// SIMATIC S7-200 SMART project (STEP 7-Micro/WIN SMART), CPU SR30

SYMBOL_TABLE M区域
自动启停1            M0.0
手动模式1            M0.1
自动模式1            M0.2
顺序启中间1           M0.3
顺序停中间1           M0.4
自动运行状态1          M0.5
故障复位1            M0.6
自动启停2            M1.0
手动模式2            M1.1
自动模式2            M1.2
顺序启中间2           M1.3
顺序停中间2           M1.4
自动运行状态2          M1.5
故障复位2            M1.6
自动启停3            M2.0
手动模式3            M2.1
自动模式3            M2.2
顺序启中间3           M2.3
顺序停中间3           M2.4
自动运行状态3          M2.5
故障复位3            M2.6
自动启停4            M3.0     // 手动按钮启
手动模式4            M3.1
自动模式4            M3.2
顺序启中间4           M3.3
顺序停中间4           M3.4
自动运行状态4          M3.5
故障复位4            M3.6
自动启停5            M4.0
手动模式5            M4.1
自动模式5            M4.2
顺序启中间5           M4.3
顺序停中间5           M4.4
自动运行状态5          M4.5
故障复位5            M4.6
进料管破1SD          M5.0
进料管破2SD          M5.1
引风机SD            M5.2
脉冲仪1SD           M5.3
脉冲仪2SD           M5.4
脉冲仪3SD           M5.5
仓泵1出口阀1SD        M5.6
仓泵1出口阀2SD        M5.7
仓泵1呼吸阀SD         M6.0
仓泵1进料阀SD         M6.1
仓泵1进料阀上SD        M6.2
仓泵1仓顶阀SD         M6.3
仓泵1流化阀SD         M6.4
仓泵1输送阀SD         M6.5
仓泵2出口阀1SD        M6.6
仓泵2出口阀2SD        M6.7
仓泵2呼吸阀SD         M7.0
仓泵2进料阀SD         M7.1
仓泵2进料阀上SD        M7.2
仓泵2仓顶阀SD         M7.3
仓泵2流化阀SD         M7.4
仓泵2输送阀SD         M7.5
向上游要料信号1SD       M7.6
向上游要料信号2SD       M7.7
人工抽料阀SD          M9.0
人工抽料通风阀SD        M9.1
人工抽料进口阀1SD       M9.2
人工抽料进口阀2SD       M9.3
人工抽料进口阀3SD       M9.4
人工负压风机SD         M9.5
进料管破1ZD          M15.0    // 自动标志
进料管破2ZD          M15.1
引风机ZD            M15.2
仓泵1出口阀1ZD        M15.6
仓泵1出口阀2ZD        M15.7
仓泵1呼吸阀ZD         M16.0
仓泵1进料阀ZD         M16.1
仓泵1进料阀上ZD        M16.2
仓泵1仓顶阀ZD         M16.3
仓泵1流化阀ZD         M16.4
仓泵1输送阀ZD         M16.5
仓泵2出口阀1ZD        M16.6
仓泵2出口阀2ZD        M16.7
仓泵2呼吸阀ZD         M17.0
仓泵2进料阀ZD         M17.1
仓泵2进料阀上ZD        M17.2
仓泵2仓顶阀ZD         M17.3
仓泵2流化阀ZD         M17.4
仓泵2输送阀ZD         M17.5
仓泵3出口阀1ZD        M17.6
仓泵3出口阀ZD         M17.7
仓泵3呼吸阀ZD         M18.0
仓泵3进料阀ZD         M18.1
仓泵3进料阀上ZD        M18.2
仓泵3仓顶阀ZD         M18.3
仓泵3流化阀ZD         M18.4
仓泵3输送阀ZD         M18.5
仓泵2出口阀ZD         M18.6
仓泵1出口阀ZD         M18.7
仓泵4出口阀ZD         M19.0
仓泵4呼吸阀ZD         M19.1
仓泵4进料阀ZD         M19.2
仓泵4进料阀上ZD        M19.3
仓泵4仓顶阀ZD         M19.4
仓泵4流化阀ZD         M19.5
仓泵4输送阀ZD         M19.6
仓泵5出口阀ZD         M19.7
仓泵5呼吸阀ZD         M20.0
仓泵5进料阀ZD         M20.1
仓泵5进料阀上ZD        M20.2
仓泵5仓顶阀ZD         M20.3
仓泵5流化阀ZD         M20.4
仓泵5输送阀ZD         M20.5
进口阀1ZD           M21.0
出口阀1ZD           M21.1
脉冲仪1ZD           M21.2
进口阀2ZD           M21.3
出口阀2ZD           M21.4
脉冲仪2ZD           M21.5
进口阀3ZD           M21.6
出口阀3ZD           M21.7
脉冲仪3ZD           M22.0
进口阀4ZD           M22.1
出口阀4ZD           M22.2
脉冲仪4ZD           M22.3
许可按钮             M25.0
除尘器切换中           M25.7
除尘器1剔除           M26.0
除尘器2剔除           M26.1
除尘器3剔除           M26.2
除尘器4剔除           M26.3
仓泵1进料            M27.0
仓泵1出料            M27.1
仓泵1等待            M27.2
仓泵2进料            M27.3
仓泵2出料            M27.4
仓泵2等待            M27.5
仓泵3进料            M27.6
仓泵3出料            M27.7
仓泵3等待            M28.0
仓泵4进料            M28.1
仓泵4出料            M28.2
仓泵4等待            M28.3
仓泵5进料            M28.4
仓泵5出料            M28.5
仓泵5等待            M28.6
累计时间复位           M29.7
风机切换按钮           M30.0
风机切换状态           M30.1
除尘器1运行           V0.0
除尘器1停止           V0.1
除尘器1满料           V0.2
除尘器1禁止进料         V0.3
进口阀1ZJ           V0.4
出口阀1ZJ           V0.5
脉冲仪1ZJ           V0.6
仓泵禁止切换1          V0.7
除尘器2运行           V1.0
除尘器2停止           V1.1
除尘器2满料           V1.2
除尘器2禁止进料         V1.3
进口阀2ZJ           V1.4
出口阀2ZJ           V1.5
脉冲仪2ZJ           V1.6
仓泵禁止切换2          V1.7
除尘器3运行           V2.0
除尘器3停止           V2.1
除尘器3满料           V2.2
除尘器3禁止进料         V2.3
进口阀3ZJ           V2.4
出口阀3ZJ           V2.5
脉冲仪3ZJ           V2.6
仓泵禁止切换3          V2.7
除尘器4运行           V3.0
除尘器4停止           V3.1
除尘器4满料           V3.2
除尘器4禁止进料         V3.3
进口阀4ZJ           V3.4
出口阀4ZJ           V3.5
脉冲仪4ZJ           V3.6
仓泵禁止切换4          V3.7
仓泵1出口阀ZJ         V5.0
仓泵1呼吸阀ZJ         V5.1
仓泵1进料阀ZJ         V5.2
仓泵1进料阀上ZJ        V5.3
仓泵1仓顶阀ZJ         V5.4
仓泵1流化阀ZJ         V5.5
仓泵1输送阀ZJ         V5.6
仓泵1禁止输送          V5.7
仓泵2出口阀ZJ         V6.0
仓泵2呼吸阀ZJ         V6.1
仓泵2进料阀ZJ         V6.2
仓泵2进料阀上ZJ        V6.3
仓泵2仓顶阀ZJ         V6.4
仓泵2流化阀ZJ         V6.5
仓泵2输送阀ZJ         V6.6
仓泵2禁止输送          V6.7
仓泵3出口阀ZJ         V7.0
仓泵3呼吸阀ZJ         V7.1
仓泵3进料阀ZJ         V7.2
仓泵3进料阀上ZJ        V7.3
仓泵3仓顶阀ZJ         V7.4
仓泵3流化阀ZJ         V7.5
仓泵3输送阀ZJ         V7.6
仓泵3禁止输送          V7.7
仓泵4出口阀ZJ         V8.0
仓泵4呼吸阀ZJ         V8.1
仓泵4进料阀ZJ         V8.2
仓泵4进料阀上ZJ        V8.3
仓泵4仓顶阀ZJ         V8.4
仓泵4流化阀ZJ         V8.5
仓泵4输送阀ZJ         V8.6
仓泵4禁止输送          V8.7
仓泵5出口阀ZJ         V9.0
仓泵5呼吸阀ZJ         V9.1
仓泵5进料阀ZJ         V9.2
仓泵5进料阀上ZJ        V9.3
仓泵5仓顶阀ZJ         V9.4
仓泵5流化阀ZJ         V9.5
仓泵5输送阀ZJ         V9.6
仓泵5禁止输送          V9.7
急停故障M            V15.0    // 急停故障 系统1
急停_V             V15.1
                 V17.0    // 系统2
                 V18.0    // 系统3
系统3总故障M          V19.5
系统2总故障M          V19.6
系统1总故障M          V19.7
AI1_ER0          V20.0    // 系统1报警
AI1_ER1          V20.1
AI1_ER2          V20.2
AI1_ER3          V20.3
AI1_ER4          V20.4
AI1_ER5          V20.5
AI1_ER6          V20.6
AI1_ER7          V20.7
AI2_ER0          V21.0    // 系统2报警
AI2_ER1          V21.1
AI2_ER2          V21.2
AI2_ER3          V21.3
AI2_ER4          V21.4
AI2_ER5          V21.5
AI2_ER6          V21.6
AI2_ER7          V21.7
AI3_ER0          V22.0    // 系统3报警
AI3_ER1          V22.1
AI3_ER2          V22.2
AI3_ER3          V22.3
AI3_ER4          V22.4
AI3_ER5          V22.5
AI3_ER6          V22.6
AI3_ER7          V22.7
AI4_ER0          V23.0    // 备用报警
AI4_ER1          V23.1
AI4_ER2          V23.2
AI4_ER3          V23.3
AI4_ER4          V23.4
AI4_ER5          V23.5
AI4_ER6          V23.6
AI4_ER7          V23.7
AI1_ST0          V24.0    // 系统1报警
AI1_ST1          V24.1
AI1_ST2          V24.2
AI1_ST3          V24.3
AI1_ST4          V24.4
AI1_ST5          V24.5
AI1_ST6          V24.6
AI1_ST7          V24.7
AI2_ST0          V25.0    // 系统2报警
AI2_ST1          V25.1
AI2_ST2          V25.2
AI2_ST3          V25.3
AI2_ST4          V25.4
AI2_ST5          V25.5
AI2_ST6          V25.6
AI2_ST7          V25.7
AI3_ST0          V26.0    // 系统3报警
AI3_ST1          V26.1
AI3_ST2          V26.2
AI3_ST3          V26.3
AI3_ST4          V26.4
AI3_ST5          V26.5
AI3_ST6          V26.6
AI3_ST7          V26.7
AI4_ST0          V27.0    // 备用报警
AI4_ST1          V27.1
AI4_ST2          V27.2
AI4_ST3          V27.3
AI4_ST4          V27.4
AI4_ST5          V27.5
AI4_ST6          V27.6
AI4_ST7          V27.7
END_SYMBOL_TABLE

SYMBOL_TABLE 系统符号
Always_On        SM0.0    // 始终接通
First_Scan_On    SM0.1    // 仅在第一个扫描周期时接通
Clock_1s         SM0.5    // 针对 1 s 的周期时间，时钟脉冲接通 0.5 s，断开 0.5 s.
END_SYMBOL_TABLE

SYMBOL_TABLE V区域
Time1            VW200
Time2            VW202
Time3            VW204
Time4            VW206
Time5            VW208
Time6            VW210
Time7            VW212
Time8            VW214
Time9            VW216
Time10           VW218
Time11           VW220
Time12           VW222
Time13           VW224
Time14           VW226
Time15           VW228
Time16           VW230
Time17           VW232
Time18           VW234
Time19           VW236
Time20           VW238
Time21           VW240
Time22           VW242
Time23           VW244
Time24           VW246
Time25           VW248
Time26           VW250
Time27           VW252
Time28           VW254
Time29           VW256
Time30           VW258
Time31           VW260
Time32           VW262
Time33           VW264
Time34           VW266
Time35           VW268
Time36           VW270
Time37           VW272
Time38           VW274
Time39           VW276
Time40           VW278
Time41           VW280
Time42           VW282
Time43           VW284
Time44           VW286
Time45           VW288
Time46           VW290
Time47           VW292
Time48           VW294
Time49           VW296
Time50           VW298
Time51           VW300
Time52           VW302
Time53           VW304
Time54           VW306
Time55           VW308
Time56           VW310
Time57           VW312
Time58           VW314
Time59           VW316
Time60           VW318
Time61           VW320
Time62           VW322
Time63           VW324
Time64           VW326
Time65           VW328
Time66           VW330
Time67           VW332
Time68           VW334
Time69           VW336
Time70           VW338
Time71           VW340
Time72           VW342
Time73           VW344
Time74           VW346
Time75           VW348
Time76           VW350
Time77           VW352
Time78           VW354
Time79           VW356
Time80           VW358
Time81           VW360
Time82           VW362
Time83           VW364
Time84           VW366
Time85           VW368
Time86           VW370
Time87           VW372
Time88           VW374
Time89           VW376
Time90           VW378
Time91           VW380
Time92           VW382
Time93           VW384
Time94           VW386
Time95           VW388
Time96           VW390
Time97           VW392
Time98           VW394
Time99           VW396
Time100          VW398
Time101          VW400
Time102          VW402
Time103          VW404
Time104          VW406
Time105          VW408
Time106          VW410
Time107          VW412
Time108          VW414
Time109          VW416
Time110          VW418
Time111          VW420
Time112          VW422
Time113          VW424
Time114          VW426
Time115          VW428
Time116          VW430
Time117          VW432
Time118          VW434
Time119          VW436
Time120          VW438
Time121          VW440
Time122          VW442
Time123          VW444
Time124          VW446
Time125          VW448
Time126          VW450
Time127          VW452
Time128          VW454
Time129          VW456
Time130          VW458
Time131          VW460
Time132          VW462
Time133          VW464
Time134          VW466
Time135          VW468
Time136          VW470
Time137          VW472
Time138          VW474
Time139          VW476
Time140          VW478
Time141          VW480
Time142          VW482
Time143          VW484
Time144          VW486
Time145          VW488
Time146          VW490
Time147          VW492
Time148          VW494
Time149          VW496
Time150          VW498
AI_Sst_L0        VD500    // 模拟量下限0
AI_Sst_L1        VD504    // 模拟量下限1
AI_Sst_L2        VD508    // 模拟量下限2
AI_Sst_L3        VD512    // 模拟量下限3
AI_Sst_L4        VD516    // 模拟量下限4
AI_Sst_L5        VD520    // 模拟量下限5
AI_Sst_L6        VD524    // 模拟量下限6
AI_Sst_L7        VD528    // 模拟量下限7
AI_Sst_L8        VD532    // 模拟量下限8
AI_Sst_L9        VD536    // 模拟量下限9
AI_Sst_L10       VD540    // 模拟量下限10
AI_Sst_L11       VD544    // 模拟量下限11
AI_Sst_L12       VD548    // 模拟量下限12
AI_Sst_L13       VD552    // 模拟量下限13
AI_Sst_L14       VD556    // 模拟量下限14
AI_Sst_L15       VD560    // 模拟量下限15
AI_Sst_L16       VD564    // 模拟量下限16
AI_Sst_L17       VD568    // 模拟量下限17
AI_Sst_L18       VD572    // 模拟量下限18
AI_Sst_L19       VD576    // 模拟量下限19
AI_Sst_L20       VD580    // 模拟量下限20
AI_Sst_L21       VD584    // 模拟量下限21
AI_Sst_L22       VD588    // 模拟量下限22
AI_Sst_L23       VD592    // 模拟量下限23
AI_Sst_L24       VD596    // 模拟量下限24
AI_Sst_H0        VD600    // 模拟量上限0
AI_Sst_H1        VD604    // 模拟量上限1
AI_Sst_H2        VD608    // 模拟量上限2
AI_Sst_H3        VD612    // 模拟量上限3
AI_Sst_H4        VD616    // 模拟量上限4
AI_Sst_H5        VD620    // 模拟量上限5
AI_Sst_H6        VD624    // 模拟量上限6
AI_Sst_H7        VD628    // 模拟量上限7
AI_Sst_H8        VD632    // 模拟量上限8
AI_Sst_H9        VD636    // 模拟量上限9
AI_Sst_H10       VD640    // 模拟量上限10
AI_Sst_H11       VD644    // 模拟量上限11
AI_Sst_H12       VD648    // 模拟量上限12
AI_Sst_H13       VD652    // 模拟量上限13
AI_Sst_H14       VD656    // 模拟量上限14
AI_Sst_H15       VD660    // 模拟量上限15
AI_Sst_H16       VD664    // 模拟量上限16
AI_Sst_H17       VD668    // 模拟量上限17
AI_Sst_H18       VD672    // 模拟量上限18
AI_Sst_H19       VD676    // 模拟量上限19
AI_Sst_H20       VD680    // 模拟量上限20
AI_Sst_H21       VD684    // 模拟量上限21
AI_Sst_H22       VD688    // 模拟量上限22
AI_Sst_H23       VD692    // 模拟量上限23
AI_Sst_H24       VD696    // 模拟量上限24
AI_BJ_0          VD700    // 模拟量报警0
AI_BJ_1          VD704    // 模拟量报警1
AI_BJ_2          VD708    // 模拟量报警2
AI_BJ_3          VD712    // 模拟量报警3
AI_BJ_4          VD716    // 模拟量报警4
AI_BJ_5          VD720    // 模拟量报警5
AI_BJ_6          VD724    // 模拟量报警6
AI_BJ_7          VD728    // 模拟量报警7
AI_BJ_8          VD732    // 模拟量报警8
AI_BJ_9          VD736    // 模拟量报警9
AI_BJ_10         VD740    // 模拟量报警10
AI_BJ_11         VD744    // 模拟量报警11
AI_BJ_12         VD748    // 模拟量报警12
AI_BJ_13         VD752    // 模拟量报警13
AI_BJ_14         VD756    // 模拟量报警14
AI_BJ_15         VD760    // 模拟量报警15
AI_BJ_16         VD764    // 模拟量报警16
AI_BJ_17         VD768    // 模拟量报警17
AI_BJ_18         VD772    // 模拟量报警18
AI_BJ_19         VD776    // 模拟量报警19
AI_BJ_20         VD780    // 模拟量报警20
AI_BJ_21         VD784    // 模拟量报警21
AI_BJ_22         VD788    // 模拟量报警22
AI_BJ_23         VD792    // 模拟量报警23
AI_BJ_24         VD796    // 模拟量报警24
AI_TJ_0          VD800    // 模拟量停机0
AI_TJ_1          VD804    // 模拟量停机1
AI_TJ_2          VD808    // 模拟量停机2
AI_TJ_3          VD812    // 模拟量停机3
AI_TJ_4          VD816    // 模拟量停机4
AI_TJ_5          VD820    // 模拟量停机5
AI_TJ_6          VD824    // 模拟量停机6
AI_TJ_7          VD828    // 模拟量停机7
AI_TJ_8          VD832    // 模拟量停机8
AI_TJ_9          VD836    // 模拟量停机9
AI_TJ_10         VD840    // 模拟量停机10
AI_TJ_11         VD844    // 模拟量停机11
AI_TJ_12         VD848    // 模拟量停机12
AI_TJ_13         VD852    // 模拟量停机13
AI_TJ_14         VD856    // 模拟量停机14
AI_TJ_15         VD860    // 模拟量停机15
AI_TJ_16         VD864    // 模拟量停机16
AI_TJ_17         VD868    // 模拟量停机17
AI_TJ_18         VD872    // 模拟量停机18
AI_TJ_19         VD876    // 模拟量停机19
AI_TJ_20         VD880    // 模拟量停机20
AI_TJ_21         VD884    // 模拟量停机21
AI_TJ_22         VD888    // 模拟量停机22
AI_TJ_23         VD892    // 模拟量停机23
AI_TJ_24         VD896    // 模拟量停机24
AI_OUT_0         VD900    // 模拟量输出0
AI_OUT_1         VD904    // 模拟量输出1
AI_OUT_2         VD908    // 模拟量输出2
AI_OUT_3         VD912    // 模拟量输出3
AI_OUT_4         VD916    // 模拟量输出4
AI_OUT_5         VD920    // 模拟量输出5
AI_OUT_6         VD924    // 模拟量输出6
AI_OUT_7         VD928    // 模拟量输出7
AI_OUT_8         VD932    // 模拟量输出8
AI_OUT_9         VD936    // 模拟量输出9
AI_OUT_10        VD940    // 模拟量输出10
AI_OUT_11        VD944    // 模拟量输出11
AI_OUT_12        VD948    // 模拟量输出12
AI_OUT_13        VD952    // 模拟量输出13
AI_OUT_14        VD956    // 模拟量输出14
AI_OUT_15        VD960    // 模拟量输出15
AI_OUT_16        VD964    // 模拟量输出16
AI_OUT_17        VD968    // 模拟量输出17
AI_OUT_18        VD972    // 模拟量输出18
AI_OUT_19        VD976    // 模拟量输出19
AI_OUT_20        VD980    // 模拟量输出20
AI_OUT_21        VD984    // 模拟量输出21
AI_OUT_22        VD988    // 模拟量输出22
AI_OUT_23        VD992    // 模拟量输出23
AI_OUT_24        VD996    // 模拟量输出24
Set_INT_0        VW1000   // 一般整数设置
Set_INT_1        VW1002
Set_INT_2        VW1004
Set_INT_3        VW1006
Set_INT_4        VW1008
Set_INT_5        VW1010
Set_INT_6        VW1012
Set_INT_7        VW1014
Set_INT_8        VW1016
Set_INT_9        VW1018
Set_INT_10       VW1020
Set_INT_11       VW1022
Set_INT_12       VW1024
Set_INT_13       VW1026
Set_INT_14       VW1028
Out_INT_0        VW1030   // 一般整数反馈
Out_INT_1        VW1032
Out_INT_2        VW1034
Out_INT_3        VW1036
Out_INT_4        VW1038
Out_INT_5        VW1040
Out_INT_6        VW1042
Out_INT_7        VW1044
Out_INT_8        VW1046
Out_INT_9        VW1048
Out_INT_10       VW1050   // 一般整数反馈
Out_INT_11       VW1052
Out_INT_12       VW1054
Out_INT_13       VW1056
Out_INT_14       VW1058
Time_S0          VW1070   // 系统累计运行时间
Time_M0          VW1072
Time_H0          VW1074
Time_D0          VW1076
Time_S1          VW1078
Time_M1          VW1080
Time_H1          VW1082
Time_D1          VW1084
Time_S2          VW1086
Time_M2          VW1088
Time_H2          VW1090
Time_D2          VW1092
Set_R0           VD1400   // 浮点型设定
Set_R1           VD1404
Set_R2           VD1408
Set_R3           VD1412
Set_R4           VD1416
Set_R5           VD1420
Set_R6           VD1424
Set_R7           VD1428
Set_R8           VD1432
Set_R9           VD1436
Set_R10          VD1440
Set_R11          VD1444
Set_R12          VD1448
Set_R13          VD1452
Set_R14          VD1456
Set_R15          VD1460
Set_R16          VD1464
Set_R17          VD1468
Set_R18          VD1472
Set_R19          VD1476
Set_R20          VD1480
Set_R21          VD1484
Set_R22          VD1488
Set_R23          VD1492
Set_R24          VD1496
Out_R0           VD1500   // 浮点型反馈
Out_R1           VD1504
Out_R2           VD1508
Out_R3           VD1512
Out_R4           VD1516
Out_R5           VD1520
Out_R6           VD1524
Out_R7           VD1528
Out_R8           VD1532
Out_R9           VD1536
Out_R10          VD1540
Out_R11          VD1544
Out_R12          VD1548
Out_R13          VD1552
Out_R14          VD1556
Out_R15          VD1560
Out_R16          VD1564
Out_R17          VD1568
Out_R18          VD1572
Out_R19          VD1576
Out_R20          VD1580
Out_R21          VD1584
Out_R22          VD1588
Out_R23          VD1592
Out_R24          VD1596
仓泵1压力低于          VD1600
仓泵2压力低于          VD1604
仓泵3压力低于          VD1608
仓泵4压力低于          VD1612
仓泵5压力低于          VD1616
除尘器1切换值          VD1620
除尘器2切换值          VD1624
除尘器3切换值          VD1628
除尘器4切换值          VD1632
除尘器5切换值          VD1636
称重1切换值           VD1640
称重2切换值           VD1644
称重3切换值           VD1648
称重4切换值           VD1652
称重5切换值           VD1656
除尘器1设定时间         VW1660
除尘器2设定时间         VW1662
除尘器3设定时间         VW1664
除尘器4设定时间         VW1666
除尘器5设定时间         VW1668
除尘器1计时           VW1670
除尘器2计时           VW1672
除尘器3计时           VW1674
除尘器4计时           VW1676
除尘器5计时           VW1678
反打1设定时间          VW1680
反打2设定时间          VW1682
反打3设定时间          VW1684
反打4设定时间          VW1686
反打5设定时间          VW1688
反打1计时            VW1690
反打2计时            VW1692
反打3计时            VW1694
反打4计时            VW1696
反打5计时            VW1698
DINT0            VD1700
DINT1            VD1704
DINT2            VD1708
DINT3            VD1712
DINT4            VD1716
DINT5            VD1720
DINT6            VD1724
DINT7            VD1728
DINT8            VD1732
END_SYMBOL_TABLE

SYMBOL_TABLE TIMEOUT
延期执行             V1800.0
提前设定             V1800.1
密码确认             V1800.2
密码错误             V1800.3
强制冷却             V1800.4
到期               V1801.0
提前到期提醒           V1801.1
白天提醒             V1801.2
永久解锁             V1801.3
输入密码             VD1810   // 浮点数
年                VW1922
月                VW1924
日                VW1926
设定年              VW1930
设定月              VW1932
设定日              VW1934
延时月              VW1936
提前年              VW1940
提前月              VW1942
提前日              VW1944
END_SYMBOL_TABLE

SYMBOL_TABLE 通讯按需修改
控制字1             VW1100   // 通讯需要先给定047E 或者04FE
给定1              VW1102   // 十进制为 0~16384对应0~100%
控制字2             VW1110   // 由于地址冲突，不同的请从EXCL复制
给定2              VW1112   // 十进制为 0~16384对应0~100%
控制字3             VW1120   // 通讯需要先给定047E 或者04FE
给定3              VW1122   // 十进制为 0~16384对应0~100%
控制字4             VW1130   // 通讯需要先给定047E 或者04FE
给定4              VW1132   // 十进制为 0~16384对应0~100%
控制字5             VW1140   // 通讯需要先给定047E 或者04FE
给定5              VW1142   // 十进制为 0~16384对应0~100%
控制字6             VW1150   // 通讯需要先给定047E 或者04FE
给定6              VW1152   // 十进制为 0~16384对应0~100%
控制字7             VW1160   // 通讯需要先给定047E 或者04FE
给定7              VW1162   // 十进制为 0~16384对应0~100%
控制字8             VW1170   // 通讯需要先给定047E 或者04FE
给定8              VW1172   // 十进制为 0~16384对应0~100%
控制字9             VW1180   // 通讯需要先给定047E 或者04FE
给定9              VW1182   // 十进制为 0~16384对应0~100%
控制字10            VW1190   // 通讯需要先给定047E 或者04FE
给定10             VW1192   // 十进制为 0~16384对应0~100%
频率1              VW1200   // 小数点2位
电流1              VW1206   // 小数点2位
频率2              VW1210   // 小数点2位
电流2              VW1216   // 小数点2位
频率3              VW1220   // 小数点2位
电流3              VW1226   // 小数点2位
频率4              VW1230   // 小数点2位
电流4              VW1236   // 小数点2位
频率5              VW1240   // 小数点2位
电流5              VW1246   // 小数点2位
频率6              VW1250   // 小数点2位
电流6              VW1256   // 小数点2位
频率7              VW1260   // 小数点2位
电流7              VW1266   // 小数点2位
频率8              VW1270   // 小数点2位
电流8              VW1276   // 小数点2位
频率9              VW1280   // 小数点2位
电流9              VW1286   // 小数点2位
频率10             VW1290   // 小数点2位
电流10             VW1296   // 小数点2位
WC0              V60.0
WC1              V60.1
WC2              V60.2
WC3              V60.3
WC4              V60.4
WC5              V60.5
WC6              V60.6
WC7              V60.7
WC8              V61.0
WC9              V61.1
WC10             V61.2
WC11             V61.3
WC12             V61.4
WC13             V61.5
WC14             V61.6
WC15             V61.7
WC16             V62.0
WC17             V62.1
WC18             V62.2
WC19             V62.3
WC20             V62.4
切换信号             V62.7
END_SYMBOL_TABLE

SYMBOL_TABLE 仪表通讯
Uab_S            VD1310   // 施耐德仪表
Ubc_S            VD1314
Uac_S            VD1318
Ua_S             VD1322
Ub_S             VD1326
Uc_S             VD1330
Ia_S             VD1334
Ib_S             VD1338
Ic_S             VD1342
Pt_S             VD1346
EP_S             VD1350
Uab_Z            VD1360   // 以下为正泰
Ubc_Z            VD1364   // 以下为正泰
Uac_Z            VD1368   // 以下为正泰
Ua_Z             VD1372   // 以下为正泰
Ub_Z             VD1376   // 以下为正泰
Uc_Z             VD1380   // 以下为正泰
Ia_Z             VD1384   // 以下为正泰
Ib_Z             VD1388   // 以下为正泰
Ic_Z             VD1392   // 以下为正泰
Pt_Z             VD1396   // 以下为正泰
EP_Z             VD1354   // 以下为正泰
END_SYMBOL_TABLE

SYMBOL_TABLE SCR符号
仓泵1步序1           S0.0     // 步序1选择仓泵
仓泵1步序2           S0.1
仓泵1步序3           S0.2
仓泵1步序4           S0.3
仓泵1步序5           S0.4
仓泵1步序6           S0.5
仓泵2步序1           S1.0
仓泵2步序2           S1.1
仓泵2步序3           S1.2
仓泵2步序4           S1.3
仓泵2步序5           S1.4
仓泵2步序6           S1.5
仓泵3步序1           S2.0
仓泵3步序2           S2.1
仓泵3步序3           S2.2
仓泵3步序4           S2.3
仓泵3步序5           S2.4
仓泵3步序6           S2.5
仓泵4步序1           S3.0
仓泵4步序2           S3.1
仓泵4步序3           S3.2
仓泵4步序4           S3.3
仓泵4步序5           S3.4
仓泵4步序6           S3.5
仓泵5步序1           S4.0
仓泵5步序2           S4.1
仓泵5步序3           S4.2
仓泵5步序4           S4.3
仓泵5步序5           S4.4
仓泵5步序6           S4.5
END_SYMBOL_TABLE

ORGANIZATION_BLOCK MAIN:OB1
TITLE=
// 
BEGIN
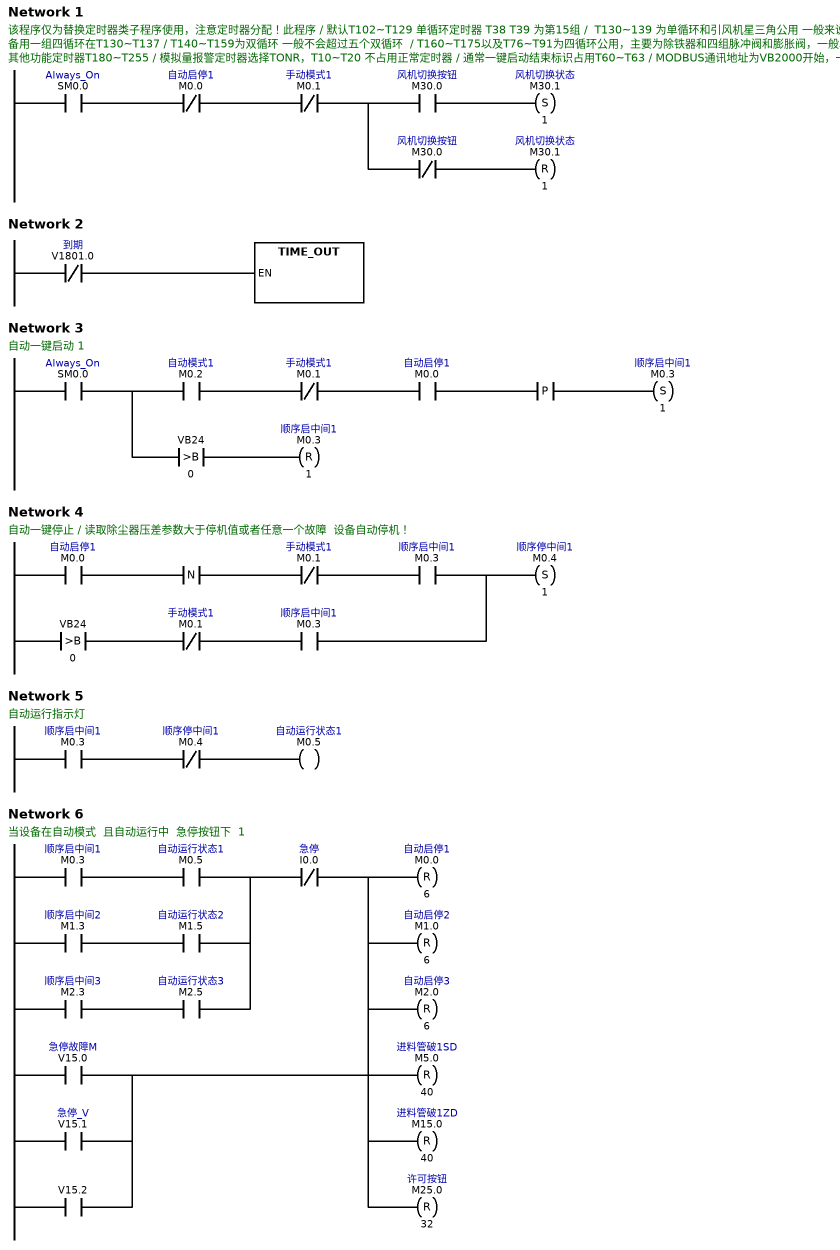
Network 1
// 该程序仅为替换定时器类子程序使用，注意定时器分配！此程序
// 默认T102~T129 单循环定时器 T38 T39 为第15组
//  T130~139 为单循环和引风机星三角公用 一般来说有星三角的程序不会用到这么多单循环阀 备用一组四循环在T130~T137
// T140~T159为双循环 一般不会超过五个双循环 
// T160~T175以及T76~T91为四循环公用，主要为除铁器和四组脉冲阀和膨胀阀，一般单独用四组
// 通常启动T40~T49 停止T50~T59 
// 其他功能定时器T180~T255
// 模拟量报警定时器选择TONR，T10~T20 不占用正常定时器
// 通常一键启动结束标识占用T60~T63
// MODBUS通讯地址为VB2000开始，一千个字节都是通讯占用区域
// 通常Time1~10为开机顺序 11~20为关机顺序 21~29为多个开关机时备用 31~80为系统仓泵或其他顺序逻辑用时间，
// Time81~120为循环时间 121~130为引风机等其他子程序时间或者循环时间备用 131~150为模拟量报警停机用
// 默认仓泵1占用T200~T214 时间31~45  仓泵2占用T215~T229 时间46~60  仓泵3占用 T230~T244 时间 61~75
// 仓泵4 占用T160~T174 时间 106~120   与四循环冲突，一般不会同时调用 与除尘器3 4 冲突
// 仓泵5占用 T175~T189 时间135~150 使用时基本会与仓泵4同时使用
// 除尘器切换主要为双除尘器 三除尘器 四除尘器 三种模式的切换子程序，只能选取一个使用
// 双除尘器切换 默认双仓泵占用 T190~T193 T46~t49  时间76~79
// 
// 
// 
LD     Always_On:SM0.0
AN     自动启停1:M0.0
AN     手动模式1:M0.1
LPS
A      风机切换按钮:M30.0
S      风机切换状态:M30.1, 1
LPP
AN     风机切换按钮:M30.0
R      风机切换状态:M30.1, 1
Network 2
LDN    到期:V1801.0
CALL   TIME_OUT:SBR5
Network 3
// 自动一键启动 1
LD     Always_On:SM0.0
LPS
A      自动模式1:M0.2
AN     手动模式1:M0.1
A      自动启停1:M0.0
EU
S      顺序启中间1:M0.3, 1
LPP
AB>    VB24, 0
R      顺序启中间1:M0.3, 1
Network 4
// 自动一键停止
// 读取除尘器压差参数大于停机值或者任意一个故障  设备自动停机！
LD     自动启停1:M0.0
ED
AN     手动模式1:M0.1
A      顺序启中间1:M0.3
LDB>   VB24, 0
AN     手动模式1:M0.1
A      顺序启中间1:M0.3
OLD
S      顺序停中间1:M0.4, 1
Network 5
// 自动运行指示灯
LD     顺序启中间1:M0.3
AN     顺序停中间1:M0.4
=      自动运行状态1:M0.5
Network 6
// 当设备在自动模式  且自动运行中  急停按钮下  1
LD     顺序启中间1:M0.3
A      自动运行状态1:M0.5
LD     顺序启中间2:M1.3
A      自动运行状态2:M1.5
OLD
LD     顺序启中间3:M2.3
A      自动运行状态3:M2.5
OLD
AN     急停:I0.0
LD     急停故障M:V15.0
O      急停_V:V15.1
O      V15.2
OLD
R      自动启停1:M0.0, 6
R      自动启停2:M1.0, 6
R      自动启停3:M2.0, 6
R      进料管破1SD:M5.0, 40
R      进料管破1ZD:M15.0, 40
R      许可按钮:M25.0, 32
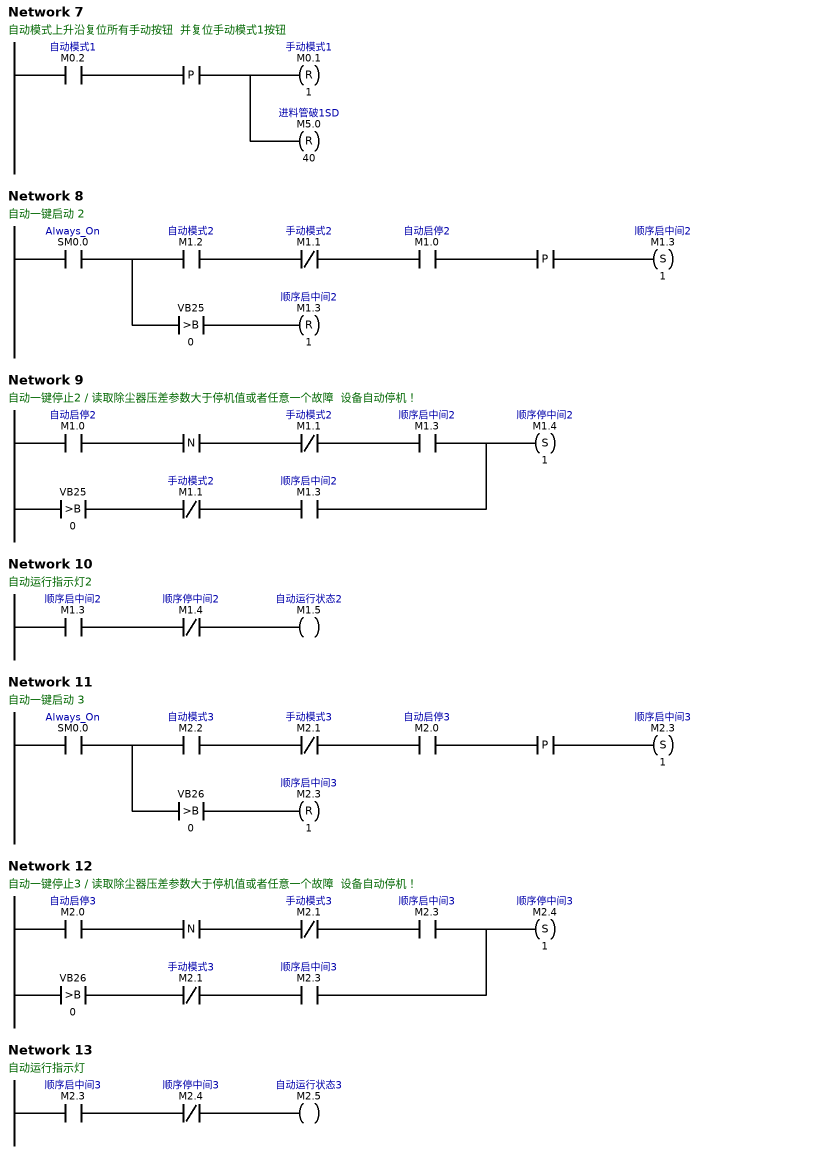
Network 7
// 自动模式上升沿复位所有手动按钮  并复位手动模式1按钮
LD     自动模式1:M0.2
EU
R      手动模式1:M0.1, 1
R      进料管破1SD:M5.0, 40
Network 8
// 自动一键启动 2
LD     Always_On:SM0.0
LPS
A      自动模式2:M1.2
AN     手动模式2:M1.1
A      自动启停2:M1.0
EU
S      顺序启中间2:M1.3, 1
LPP
AB>    VB25, 0
R      顺序启中间2:M1.3, 1
Network 9
// 自动一键停止2
// 读取除尘器压差参数大于停机值或者任意一个故障  设备自动停机！
LD     自动启停2:M1.0
ED
AN     手动模式2:M1.1
A      顺序启中间2:M1.3
LDB>   VB25, 0
AN     手动模式2:M1.1
A      顺序启中间2:M1.3
OLD
S      顺序停中间2:M1.4, 1
Network 10
// 自动运行指示灯2
LD     顺序启中间2:M1.3
AN     顺序停中间2:M1.4
=      自动运行状态2:M1.5
Network 11
// 自动一键启动 3
LD     Always_On:SM0.0
LPS
A      自动模式3:M2.2
AN     手动模式3:M2.1
A      自动启停3:M2.0
EU
S      顺序启中间3:M2.3, 1
LPP
AB>    VB26, 0
R      顺序启中间3:M2.3, 1
Network 12
// 自动一键停止3
// 读取除尘器压差参数大于停机值或者任意一个故障  设备自动停机！
LD     自动启停3:M2.0
ED
AN     手动模式3:M2.1
A      顺序启中间3:M2.3
LDB>   VB26, 0
AN     手动模式3:M2.1
A      顺序启中间3:M2.3
OLD
S      顺序停中间3:M2.4, 1
Network 13
// 自动运行指示灯
LD     顺序启中间3:M2.3
AN     顺序停中间3:M2.4
=      自动运行状态3:M2.5
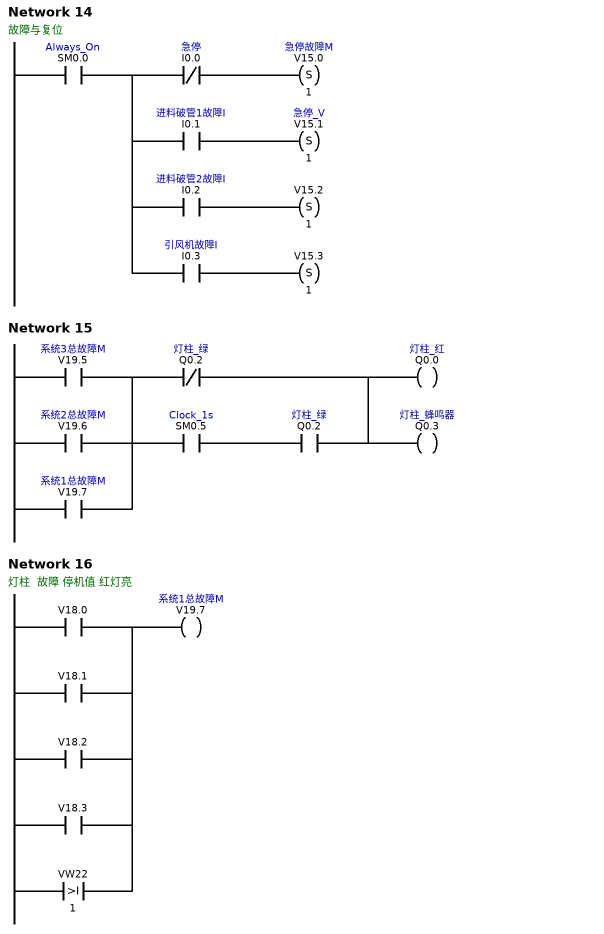
Network 14
// 故障与复位
LD     Always_On:SM0.0
LPS
AN     急停:I0.0
S      急停故障M:V15.0, 1
LRD
A      进料破管1故障I:I0.1
S      急停_V:V15.1, 1
LRD
A      进料破管2故障I:I0.2
S      V15.2, 1
LPP
A      引风机故障I:I0.3
S      V15.3, 1
Network 15
LD     系统3总故障M:V19.5
O      系统2总故障M:V19.6
O      系统1总故障M:V19.7
LDN    灯柱_绿:Q0.2
LD     Clock_1s:SM0.5
A      灯柱_绿:Q0.2
OLD
ALD
=      灯柱_红:Q0.0
=      灯柱_蜂鸣器:Q0.3
Network 16
// 灯柱  故障 停机值 红灯亮
LD     V18.0
O      V18.1
O      V18.2
O      V18.3
OW>    VW22, 1
=      系统1总故障M:V19.7
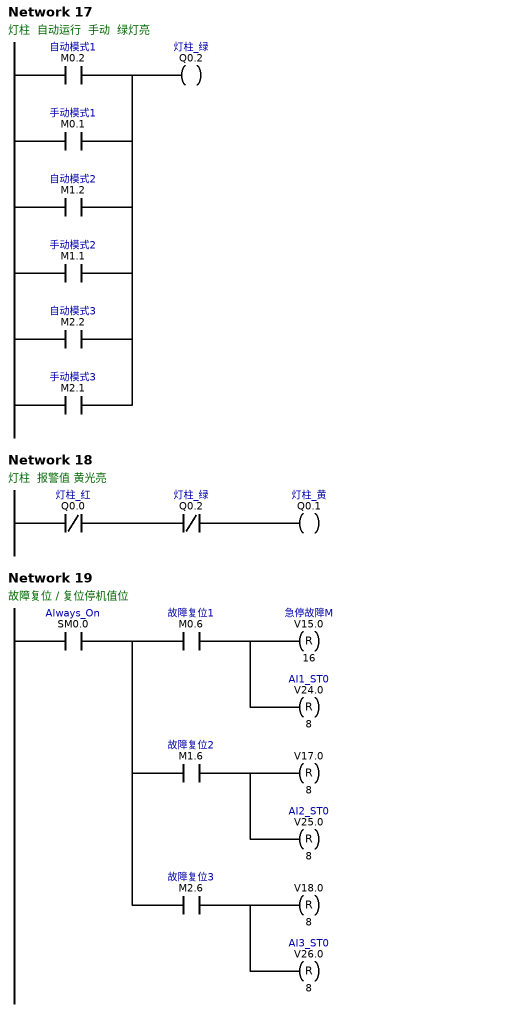
Network 17
// 灯柱  自动运行  手动  绿灯亮
LD     自动模式1:M0.2
O      手动模式1:M0.1
O      自动模式2:M1.2
O      手动模式2:M1.1
O      自动模式3:M2.2
O      手动模式3:M2.1
=      灯柱_绿:Q0.2
Network 18
// 灯柱  报警值 黄光亮
LDN    灯柱_红:Q0.0
AN     灯柱_绿:Q0.2
=      灯柱_黄:Q0.1
Network 19
// 故障复位
// 复位停机值位
LD     Always_On:SM0.0
LPS
A      故障复位1:M0.6
R      急停故障M:V15.0, 16
R      AI1_ST0:V24.0, 8
LRD
A      故障复位2:M1.6
R      V17.0, 8
R      AI2_ST0:V25.0, 8
LPP
A      故障复位3:M2.6
R      V18.0, 8
R      AI3_ST0:V26.0, 8
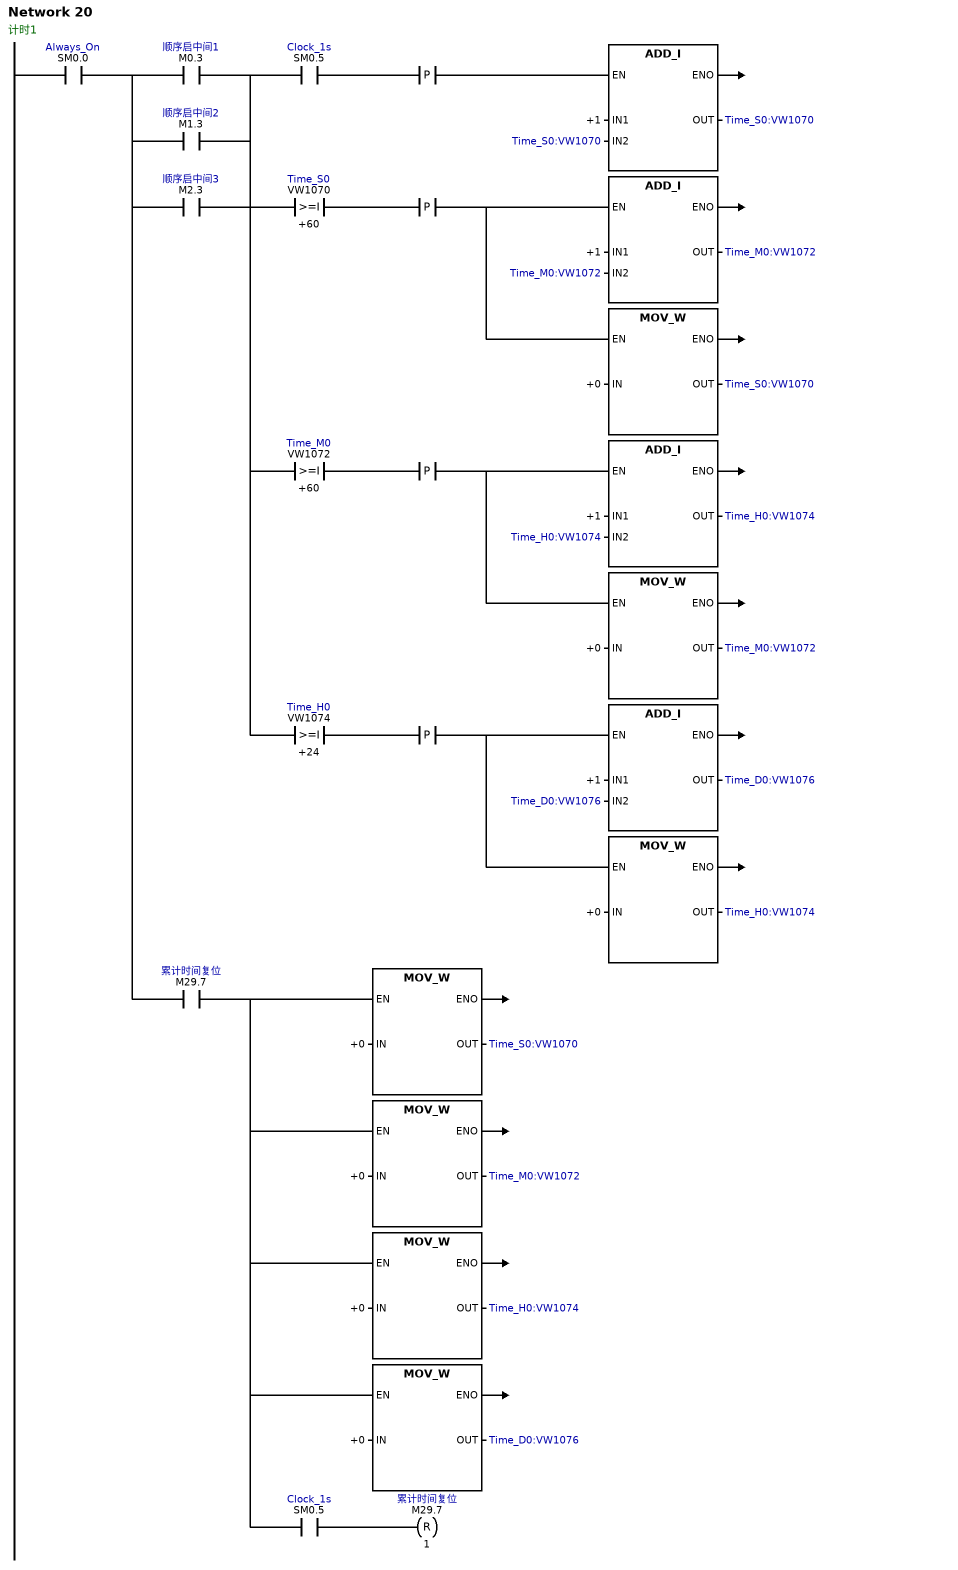
Network 20
// 计时1
LD     Always_On:SM0.0
LPS
LD     顺序启中间1:M0.3
O      顺序启中间2:M1.3
O      顺序启中间3:M2.3
ALD
LPS
A      Clock_1s:SM0.5
EU
+I     +1, Time_S0:VW1070
LRD
AW>=   Time_S0:VW1070, +60
EU
+I     +1, Time_M0:VW1072
MOVW   +0, Time_S0:VW1070
LRD
AW>=   Time_M0:VW1072, +60
EU
+I     +1, Time_H0:VW1074
MOVW   +0, Time_M0:VW1072
LPP
AW>=   Time_H0:VW1074, +24
EU
+I     +1, Time_D0:VW1076
MOVW   +0, Time_H0:VW1074
LPP
A      累计时间复位:M29.7
MOVW   +0, Time_S0:VW1070
MOVW   +0, Time_M0:VW1072
MOVW   +0, Time_H0:VW1074
MOVW   +0, Time_D0:VW1076
A      Clock_1s:SM0.5
R      累计时间复位:M29.7, 1
END_ORGANIZATION_BLOCK

// SBR0: protected block, not included

// SBR1: protected block, not included

// SBR2: protected block, not included

// SBR3: protected block, not included

// SBR4: protected block, not included

SUBROUTINE_BLOCK TIME_OUT:SBR5
TITLE=
BEGIN
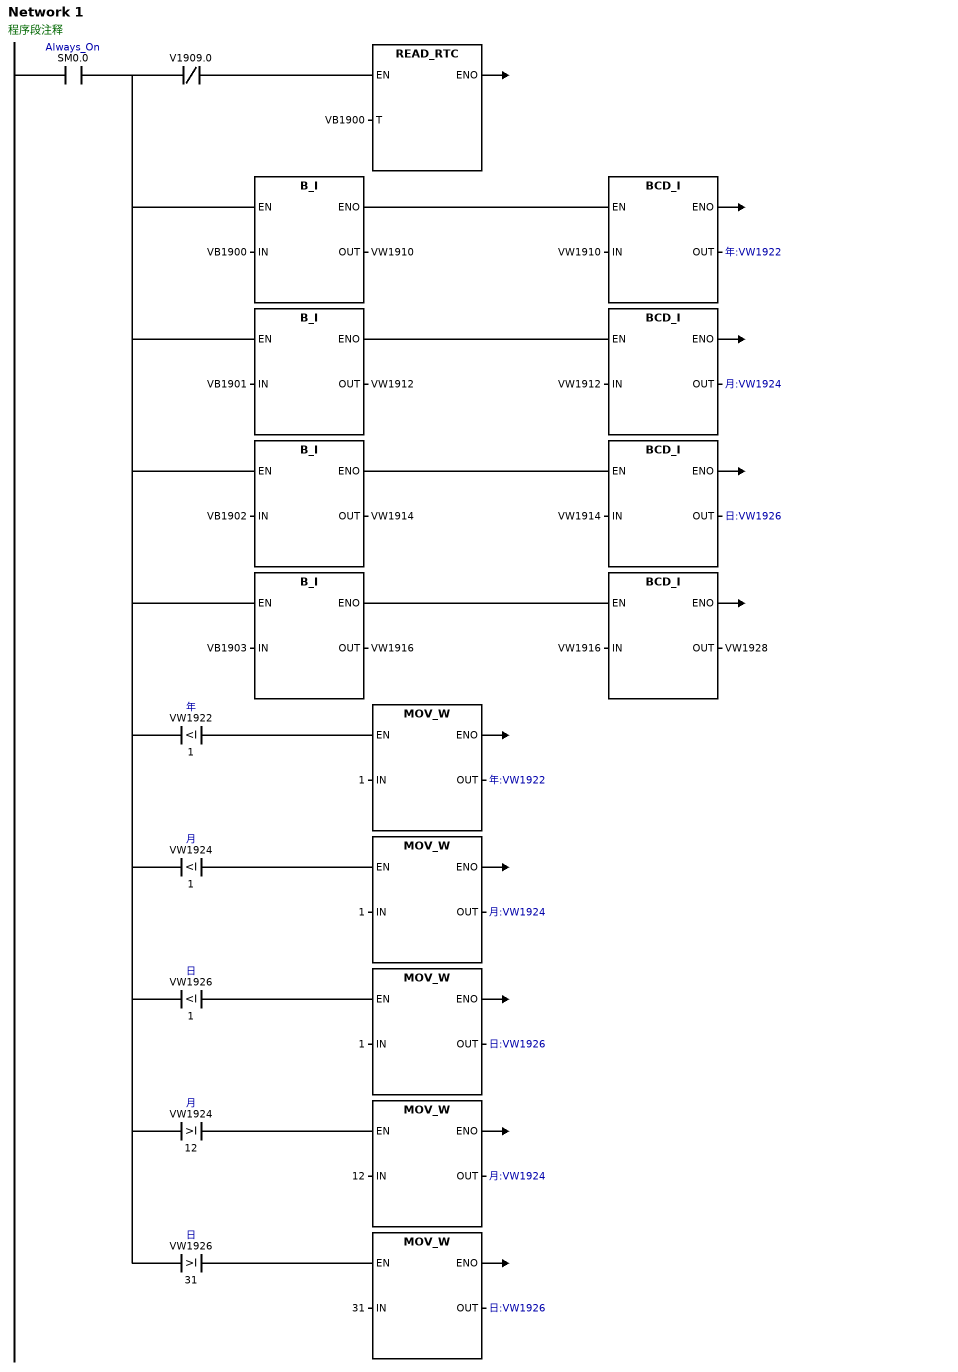
Network 1
// 程序段注释
LD     Always_On:SM0.0
LPS
AN     V1909.0
TODR   VB1900
LRD
BTI    VB1900, VW1910
AENO
MOVW   VW1910, 年:VW1922
BCDI   年:VW1922
LRD
BTI    VB1901, VW1912
AENO
MOVW   VW1912, 月:VW1924
BCDI   月:VW1924
LRD
BTI    VB1902, VW1914
AENO
MOVW   VW1914, 日:VW1926
BCDI   日:VW1926
LRD
BTI    VB1903, VW1916
AENO
MOVW   VW1916, VW1928
BCDI   VW1928
LRD
AW<    年:VW1922, 1
MOVW   1, 年:VW1922
LRD
AW<    月:VW1924, 1
MOVW   1, 月:VW1924
LRD
AW<    日:VW1926, 1
MOVW   1, 日:VW1926
LRD
AW>    月:VW1924, 12
MOVW   12, 月:VW1924
LPP
AW>    日:VW1926, 31
MOVW   31, 日:VW1926
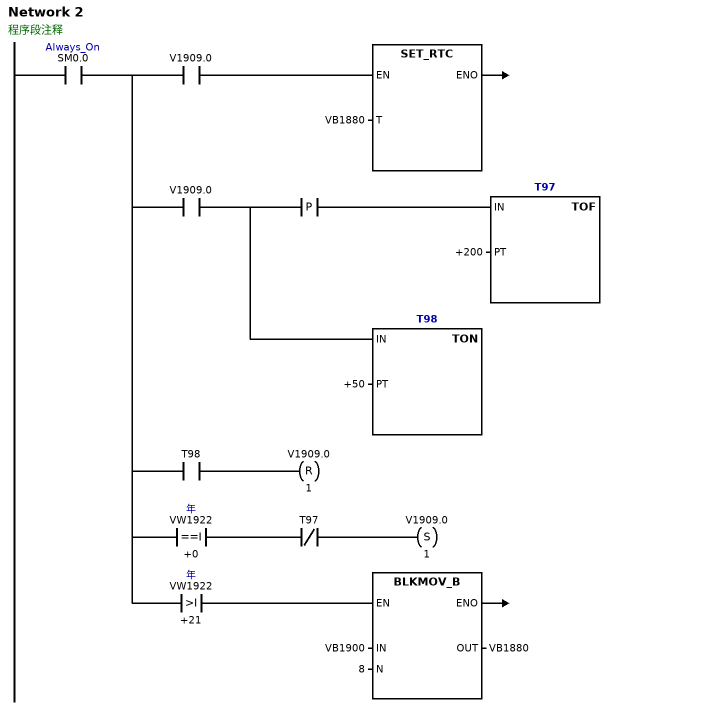
Network 2
// 程序段注释
LD     Always_On:SM0.0
LPS
A      V1909.0
TODW   VB1880
LRD
A      V1909.0
LPS
EU
TOF    T97, +200
LPP
TON    T98, +50
LPP
LPS
A      T98
R      V1909.0, 1
LRD
AW=    年:VW1922, +0
AN     T97
S      V1909.0, 1
LPP
AW>    年:VW1922, +21
BMB    VB1900, VB1880, 8
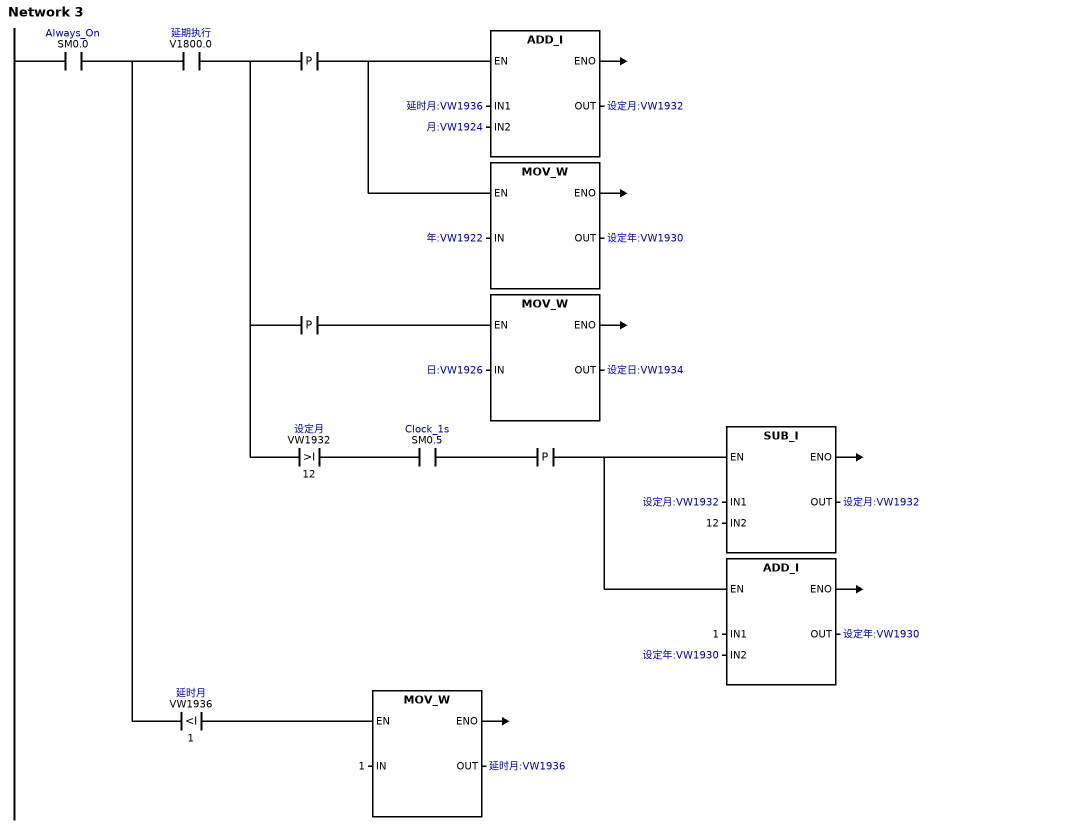
Network 3
LD     Always_On:SM0.0
LPS
A      延期执行:V1800.0
LPS
EU
MOVW   延时月:VW1936, 设定月:VW1932
+I     月:VW1924, 设定月:VW1932
MOVW   年:VW1922, 设定年:VW1930
LRD
EU
MOVW   日:VW1926, 设定日:VW1934
LPP
AW>    设定月:VW1932, 12
A      Clock_1s:SM0.5
EU
-I     12, 设定月:VW1932
+I     1, 设定年:VW1930
LPP
AW<    延时月:VW1936, 1
MOVW   1, 延时月:VW1936
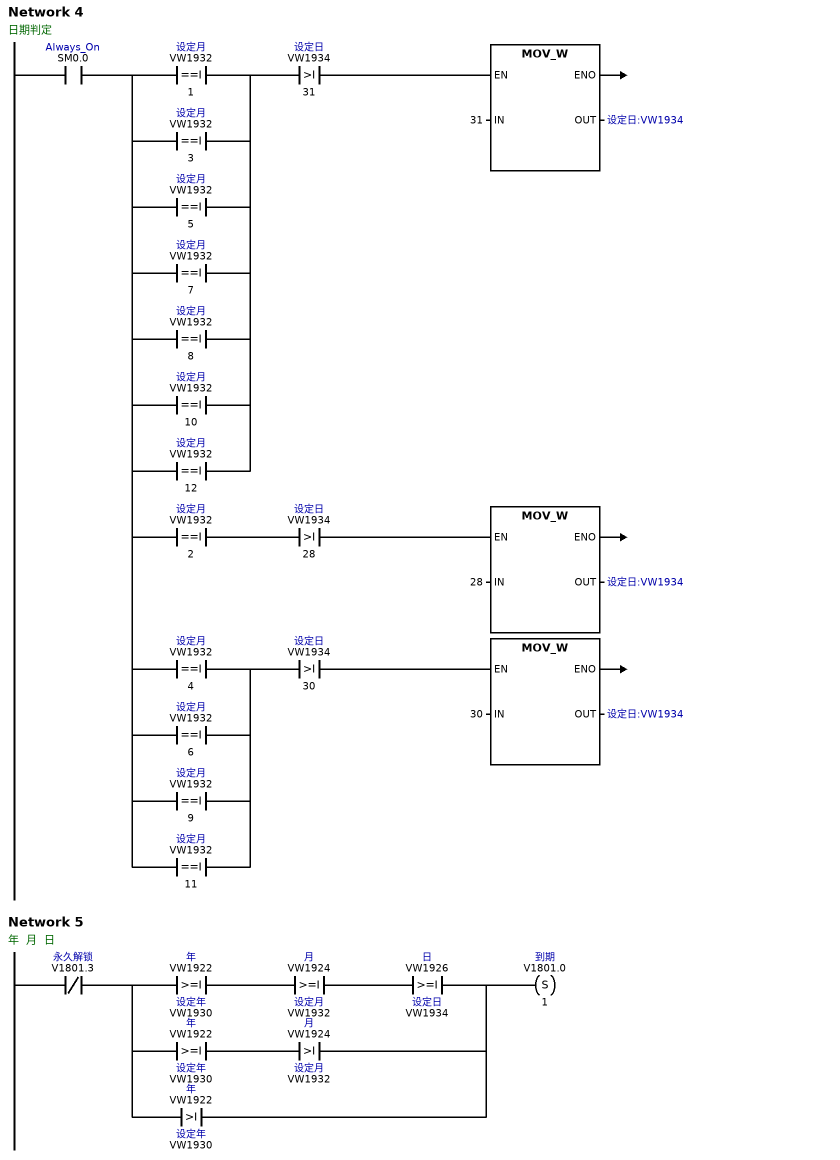
Network 4
// 日期判定
LD     Always_On:SM0.0
LPS
LDW=   设定月:VW1932, 1
OW=    设定月:VW1932, 3
OW=    设定月:VW1932, 5
OW=    设定月:VW1932, 7
OW=    设定月:VW1932, 8
OW=    设定月:VW1932, 10
OW=    设定月:VW1932, 12
ALD
AW>    设定日:VW1934, 31
MOVW   31, 设定日:VW1934
LRD
AW=    设定月:VW1932, 2
AW>    设定日:VW1934, 28
MOVW   28, 设定日:VW1934
LPP
LDW=   设定月:VW1932, 4
OW=    设定月:VW1932, 6
OW=    设定月:VW1932, 9
OW=    设定月:VW1932, 11
ALD
AW>    设定日:VW1934, 30
MOVW   30, 设定日:VW1934
Network 5
// 年  月  日 
LDN    永久解锁:V1801.3
LDW>=  年:VW1922, 设定年:VW1930
AW>=   月:VW1924, 设定月:VW1932
AW>=   日:VW1926, 设定日:VW1934
LDW>=  年:VW1922, 设定年:VW1930
AW>    月:VW1924, 设定月:VW1932
OLD
OW>    年:VW1922, 设定年:VW1930
ALD
S      到期:V1801.0, 1
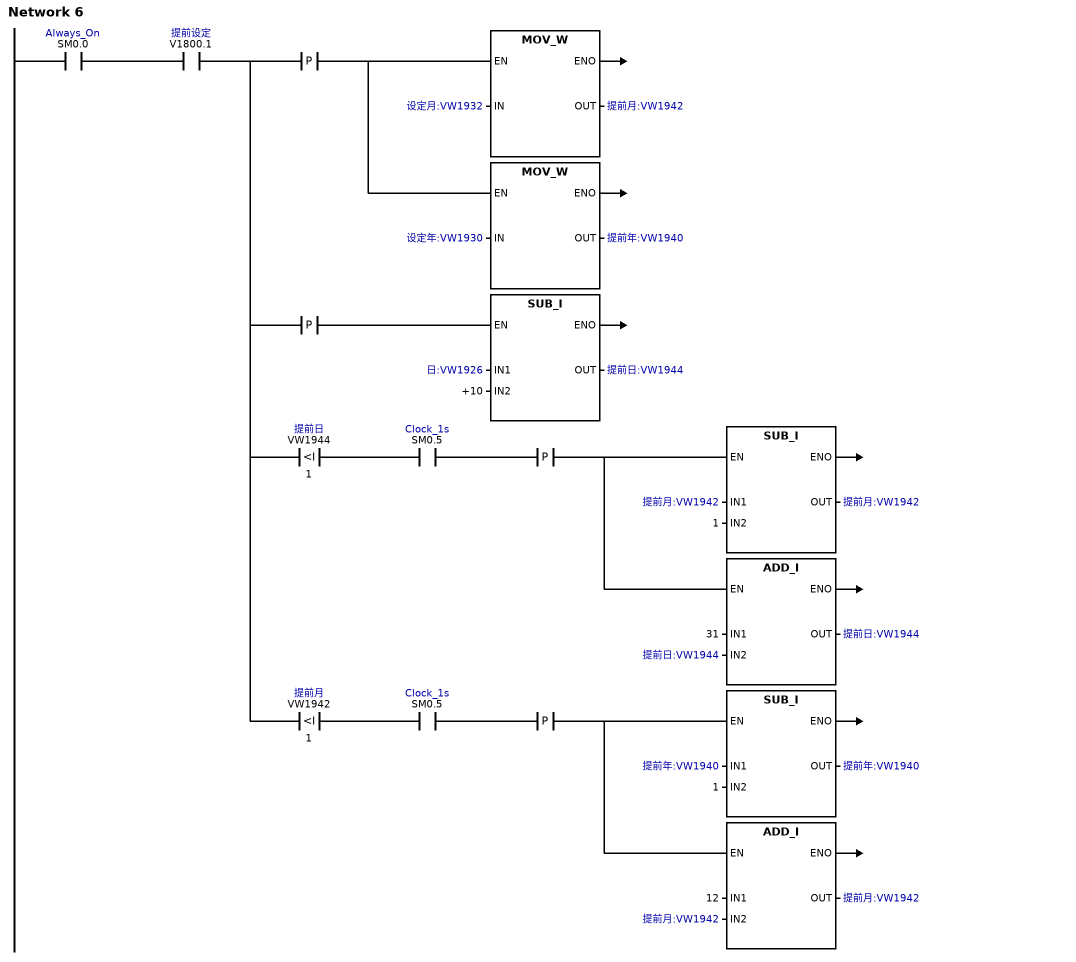
Network 6
LD     Always_On:SM0.0
A      提前设定:V1800.1
LPS
EU
MOVW   设定月:VW1932, 提前月:VW1942
MOVW   设定年:VW1930, 提前年:VW1940
LRD
EU
MOVW   日:VW1926, 提前日:VW1944
-I     +10, 提前日:VW1944
LRD
AW<    提前日:VW1944, 1
A      Clock_1s:SM0.5
EU
-I     1, 提前月:VW1942
+I     31, 提前日:VW1944
LPP
AW<    提前月:VW1942, 1
A      Clock_1s:SM0.5
EU
-I     1, 提前年:VW1940
+I     12, 提前月:VW1942
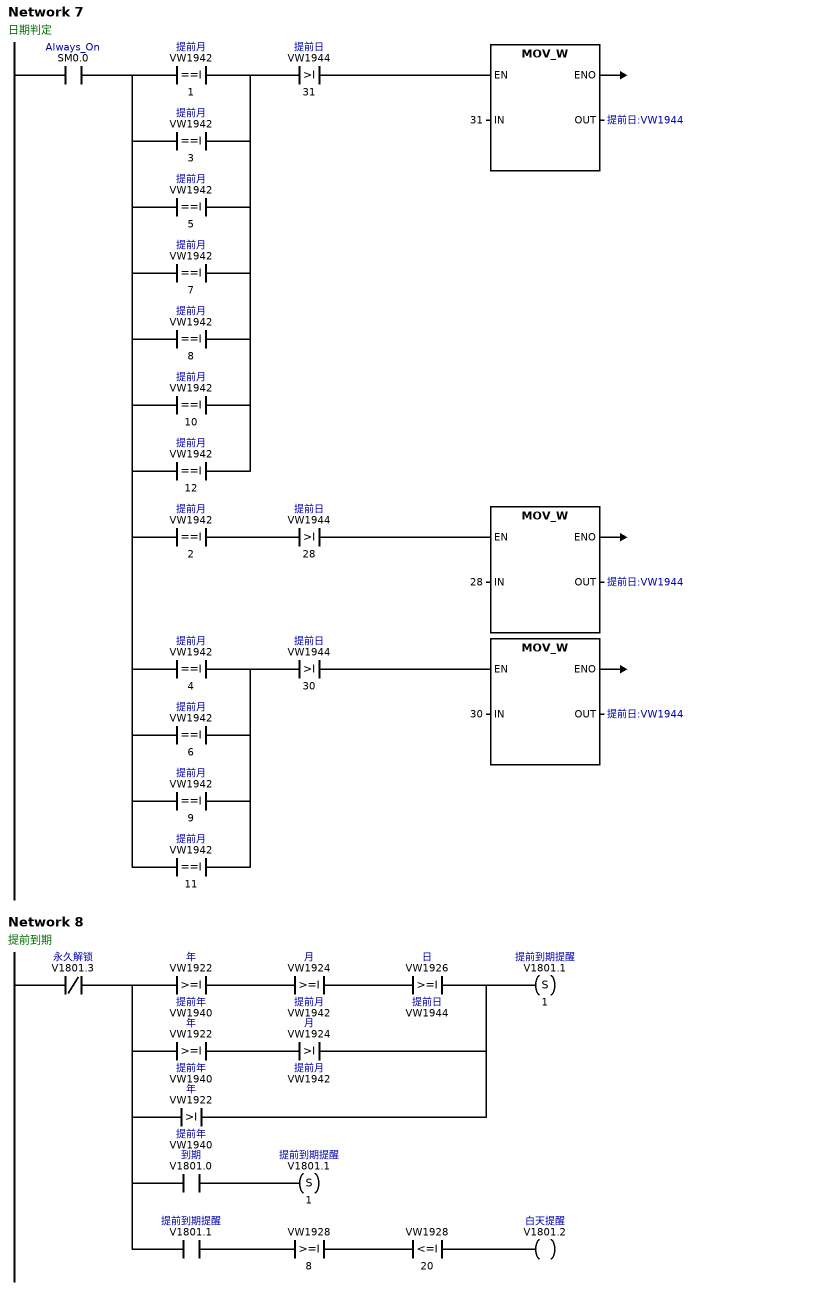
Network 7
// 日期判定
LD     Always_On:SM0.0
LPS
LDW=   提前月:VW1942, 1
OW=    提前月:VW1942, 3
OW=    提前月:VW1942, 5
OW=    提前月:VW1942, 7
OW=    提前月:VW1942, 8
OW=    提前月:VW1942, 10
OW=    提前月:VW1942, 12
ALD
AW>    提前日:VW1944, 31
MOVW   31, 提前日:VW1944
LRD
AW=    提前月:VW1942, 2
AW>    提前日:VW1944, 28
MOVW   28, 提前日:VW1944
LPP
LDW=   提前月:VW1942, 4
OW=    提前月:VW1942, 6
OW=    提前月:VW1942, 9
OW=    提前月:VW1942, 11
ALD
AW>    提前日:VW1944, 30
MOVW   30, 提前日:VW1944
Network 8
// 提前到期
LDN    永久解锁:V1801.3
LPS
LDW>=  年:VW1922, 提前年:VW1940
AW>=   月:VW1924, 提前月:VW1942
AW>=   日:VW1926, 提前日:VW1944
LDW>=  年:VW1922, 提前年:VW1940
AW>    月:VW1924, 提前月:VW1942
OLD
OW>    年:VW1922, 提前年:VW1940
ALD
S      提前到期提醒:V1801.1, 1
LPP
LPS
A      到期:V1801.0
S      提前到期提醒:V1801.1, 1
LPP
A      提前到期提醒:V1801.1
AW>=   VW1928, 8
AW<=   VW1928, 20
=      白天提醒:V1801.2
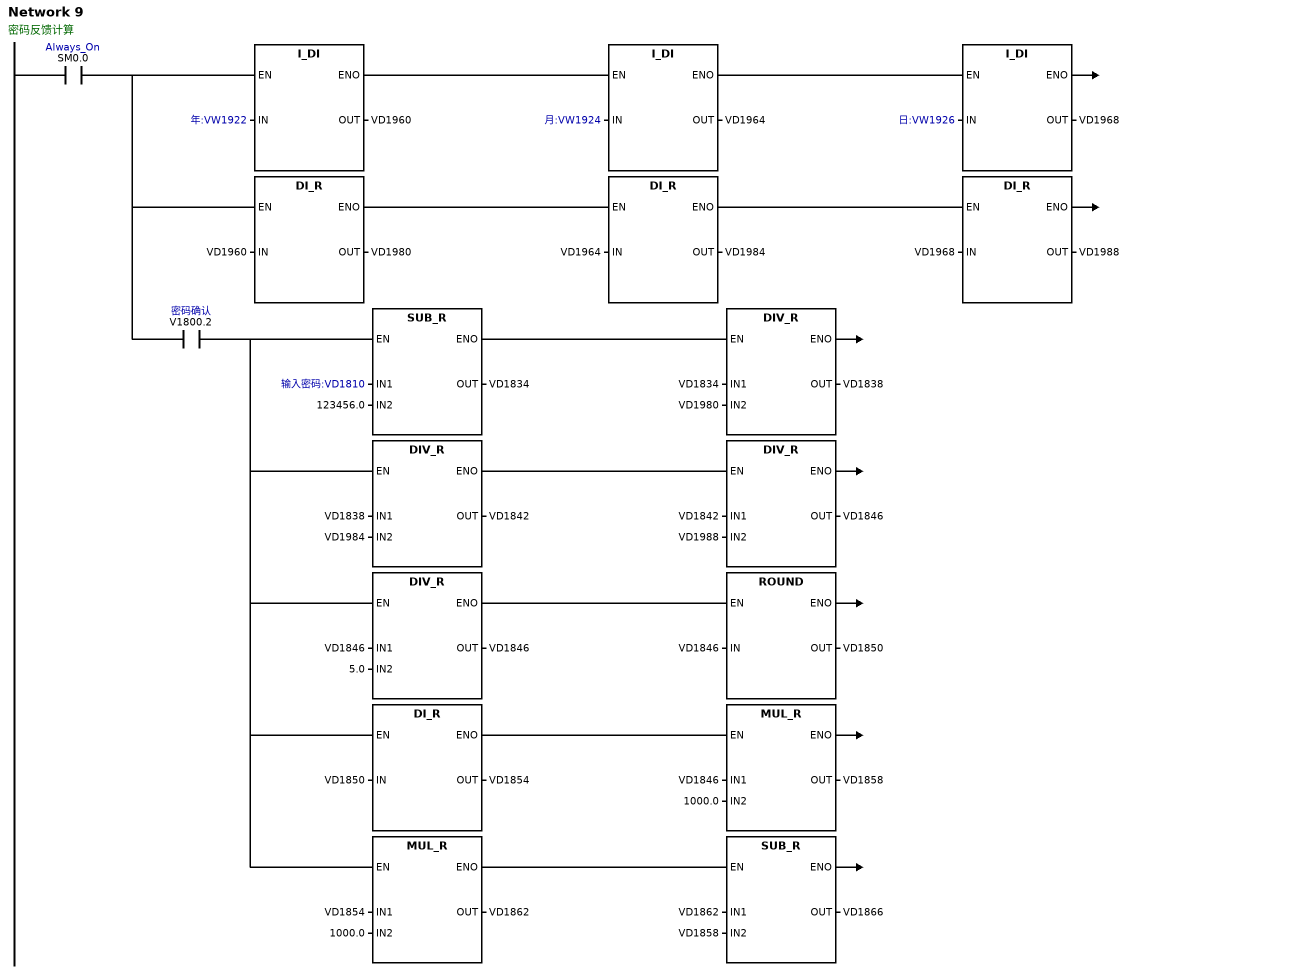
Network 9
// 密码反馈计算
LD     Always_On:SM0.0
LPS
ITD    年:VW1922, VD1960
AENO
ITD    月:VW1924, VD1964
AENO
ITD    日:VW1926, VD1968
LRD
DTR    VD1960, VD1980
AENO
DTR    VD1964, VD1984
AENO
DTR    VD1968, VD1988
LPP
A      密码确认:V1800.2
LPS
MOVR   输入密码:VD1810, VD1834
AENO
-R     123456.0, VD1834
AENO
MOVR   VD1834, VD1838
/R     VD1980, VD1838
LRD
MOVR   VD1838, VD1842
AENO
/R     VD1984, VD1842
AENO
MOVR   VD1842, VD1846
/R     VD1988, VD1846
LRD
/R     5.0, VD1846
AENO
ROUND  VD1846, VD1850
LRD
DTR    VD1850, VD1854
AENO
MOVR   VD1846, VD1858
*R     1000.0, VD1858
LPP
MOVR   VD1854, VD1862
AENO
*R     1000.0, VD1862
AENO
MOVR   VD1862, VD1866
-R     VD1858, VD1866
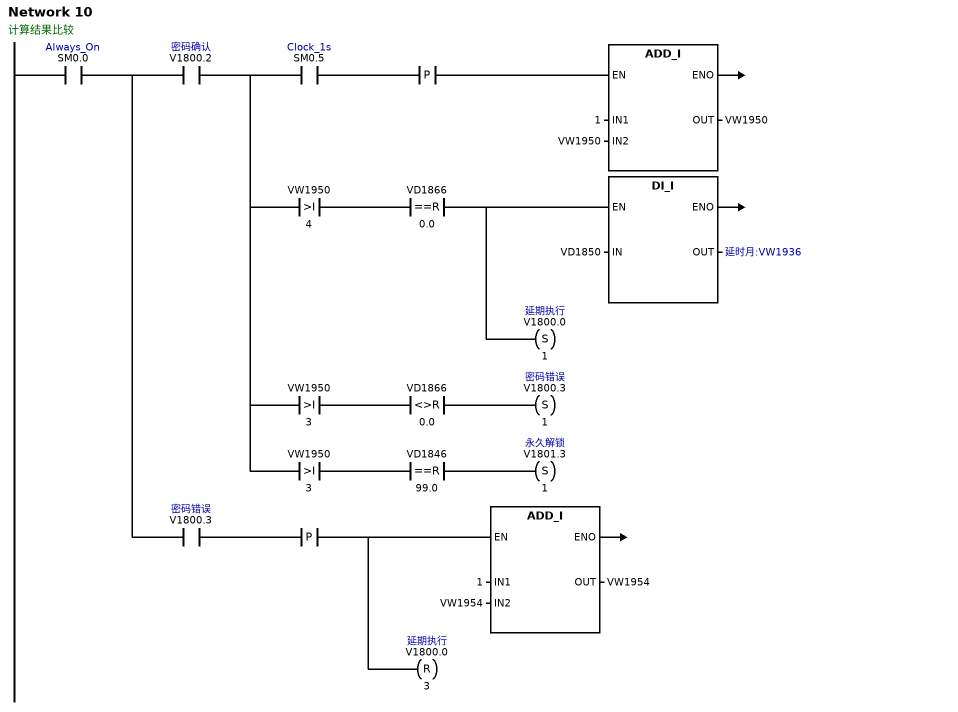
Network 10
// 计算结果比较
LD     Always_On:SM0.0
LPS
A      密码确认:V1800.2
LPS
A      Clock_1s:SM0.5
EU
+I     1, VW1950
LRD
AW>    VW1950, 4
AR=    VD1866, 0.0
DTI    VD1850, 延时月:VW1936
S      延期执行:V1800.0, 1
LPP
LPS
AW>    VW1950, 3
AR<>   VD1866, 0.0
S      密码错误:V1800.3, 1
LPP
AW>    VW1950, 3
AR=    VD1846, 99.0
S      永久解锁:V1801.3, 1
LPP
A      密码错误:V1800.3
EU
+I     1, VW1954
R      延期执行:V1800.0, 3
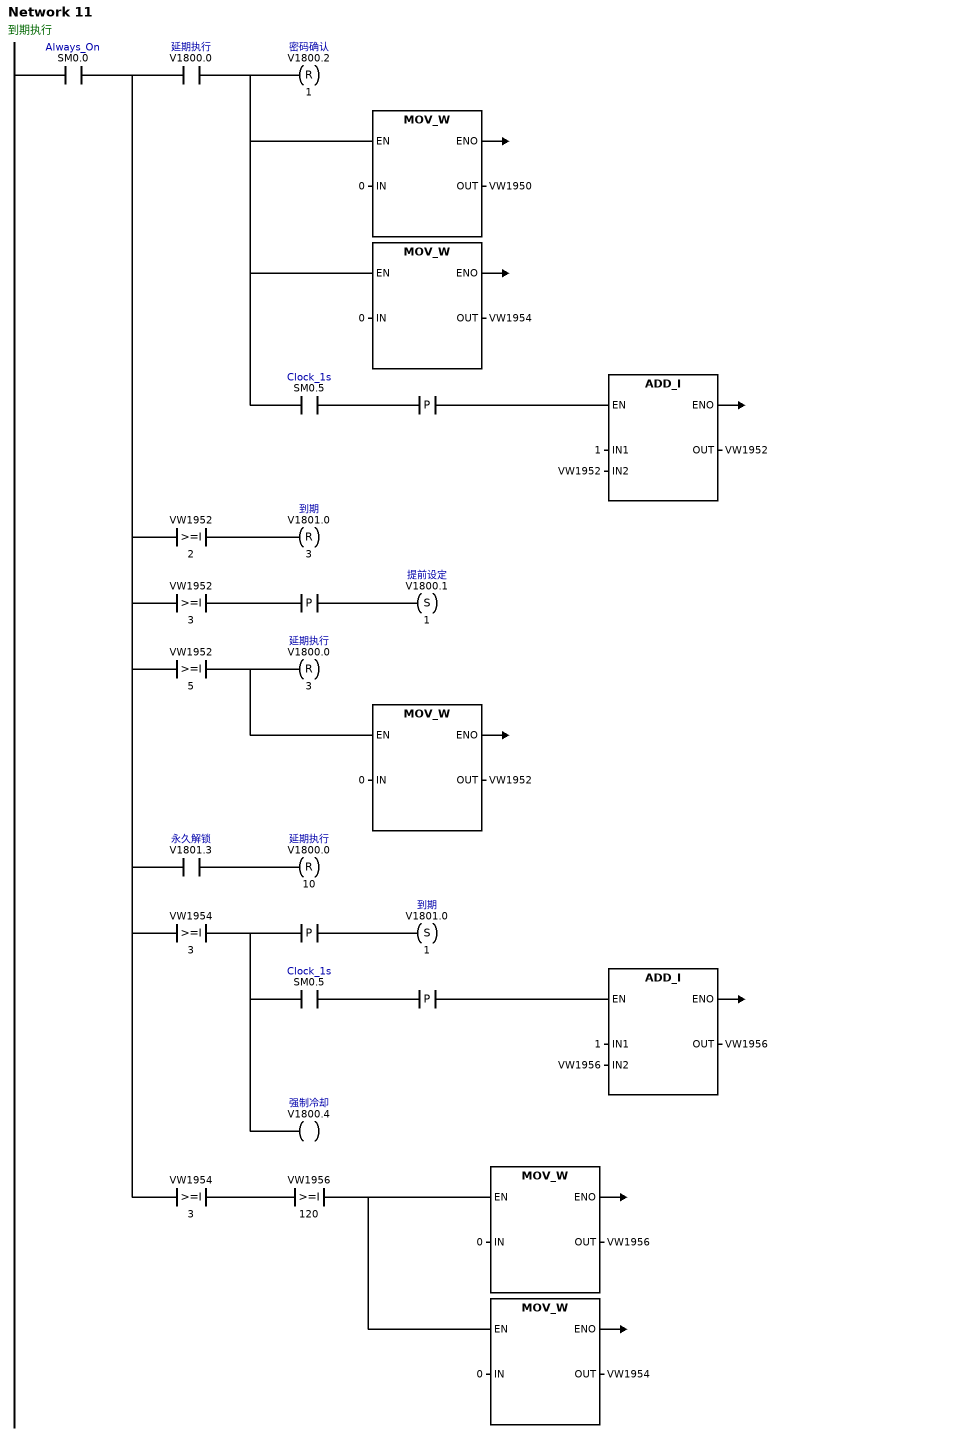
Network 11
// 到期执行
LD     Always_On:SM0.0
LPS
A      延期执行:V1800.0
R      密码确认:V1800.2, 1
MOVW   0, VW1950
MOVW   0, VW1954
A      Clock_1s:SM0.5
EU
+I     1, VW1952
LRD
LPS
AW>=   VW1952, 2
R      到期:V1801.0, 3
LPP
AW>=   VW1952, 3
EU
S      提前设定:V1800.1, 1
LRD
AW>=   VW1952, 5
R      延期执行:V1800.0, 3
MOVW   0, VW1952
LRD
A      永久解锁:V1801.3
R      延期执行:V1800.0, 10
LRD
AW>=   VW1954, 3
LPS
EU
S      到期:V1801.0, 1
LRD
A      Clock_1s:SM0.5
EU
+I     1, VW1956
LPP
=      强制冷却:V1800.4
LPP
AW>=   VW1954, 3
AW>=   VW1956, 120
MOVW   0, VW1956
MOVW   0, VW1954
END_SUBROUTINE_BLOCK

// SBR6: protected block, not included

// SBR7: protected block, not included

SUBROUTINE_BLOCK 系统按钮:SBR8
TITLE=
VAR_IN_OUT
Auto_Mode:BOOL;	// L0.0 
Hand_Mode:BOOL;	// L0.1 
System_Star:BOOL;	// L0.2 
Star_Middle:BOOL;	// L0.3 
Stop_Middle:BOOL;	// L0.4 
Auto_State:BOOL;	// L0.5 
Rest:BOOL;	// L0.6 
Standby:BOOL;	// L0.7 
Error1_Stop:BOOL;	// L1.0 
Error2_Stop:BOOL;	// L1.1 
Error3_Stop:BOOL;	// L1.2 
Error4_Stop:BOOL;	// L1.3 
System_Error:BOOL;	// L1.4 
E_Stop:BOOL;	// L1.5 
Stop_over:BOOL;	// L1.6 
END_VAR
BEGIN
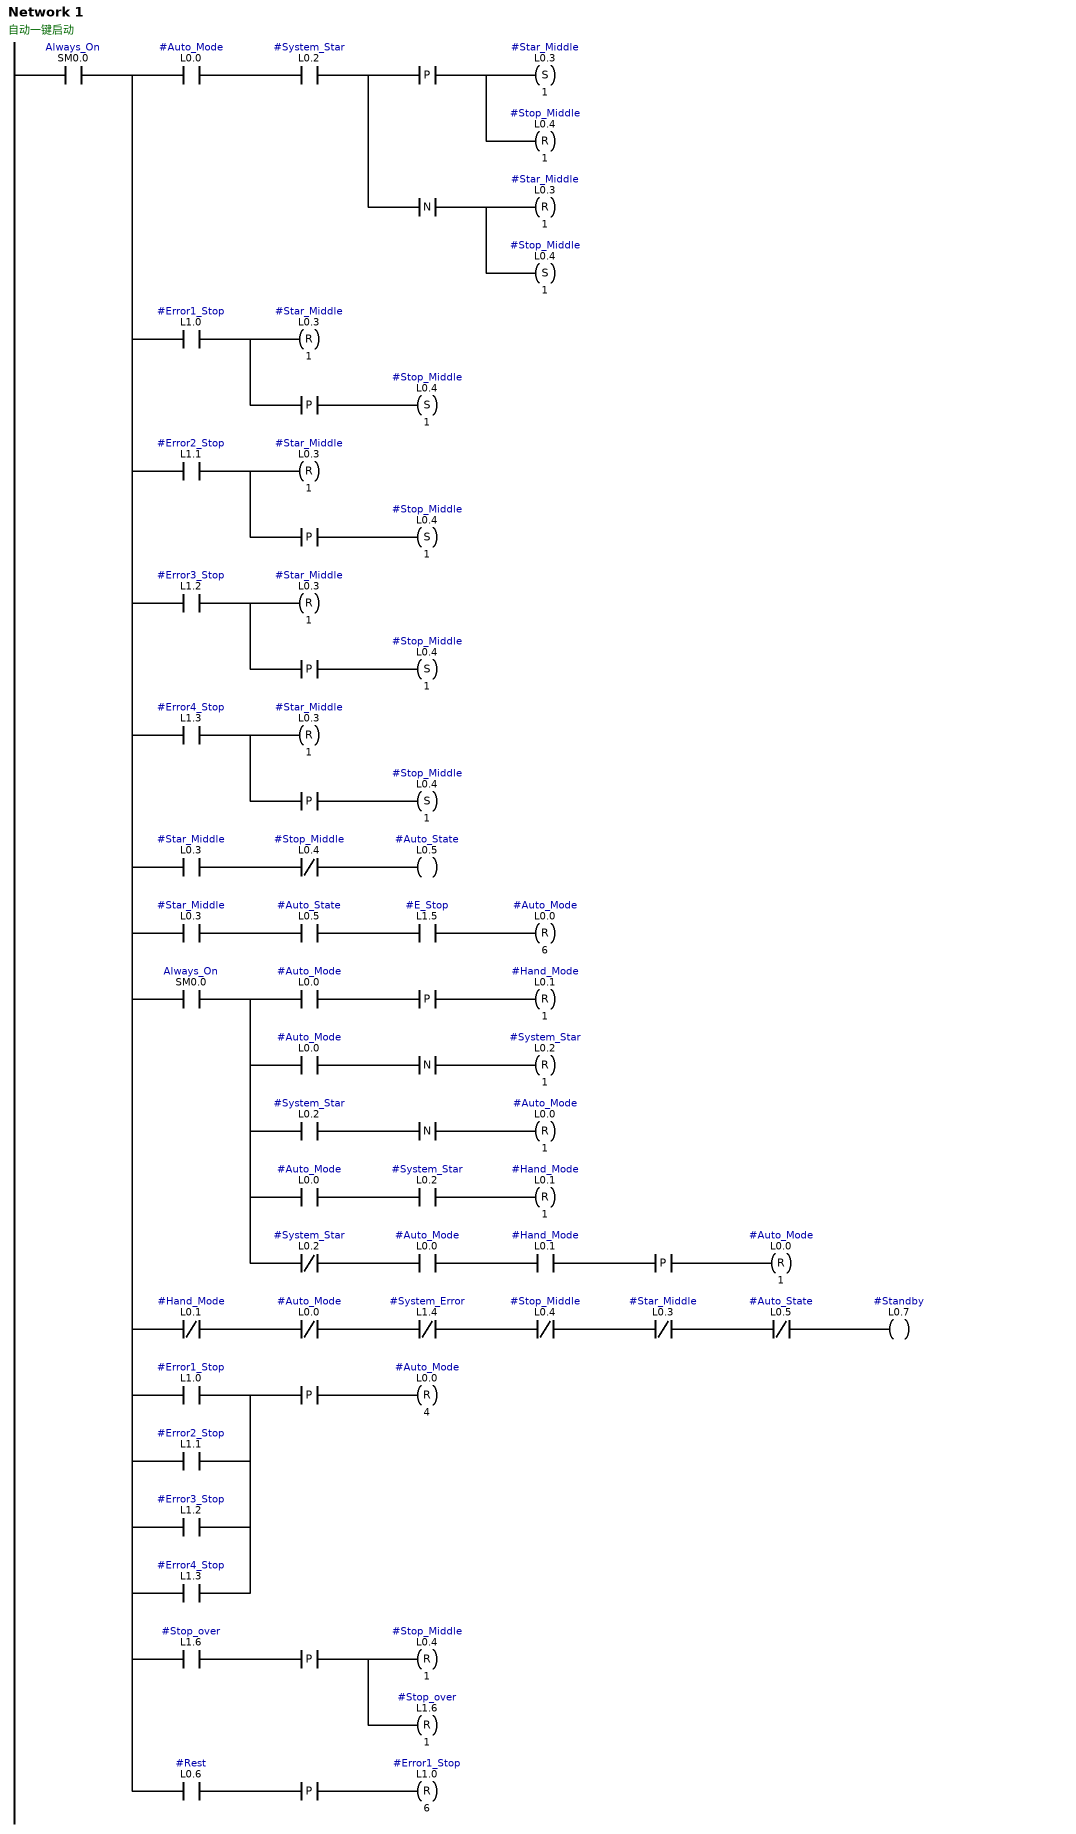
Network 1
// 自动一键启动 
LD     Always_On:SM0.0
LPS
A      #Auto_Mode:L0.0
A      #System_Star:L0.2
LPS
EU
S      #Star_Middle:L0.3, 1
R      #Stop_Middle:L0.4, 1
LPP
ED
R      #Star_Middle:L0.3, 1
S      #Stop_Middle:L0.4, 1
LPP
LPS
A      #Error1_Stop:L1.0
R      #Star_Middle:L0.3, 1
EU
S      #Stop_Middle:L0.4, 1
LRD
A      #Error2_Stop:L1.1
R      #Star_Middle:L0.3, 1
EU
S      #Stop_Middle:L0.4, 1
LRD
A      #Error3_Stop:L1.2
R      #Star_Middle:L0.3, 1
EU
S      #Stop_Middle:L0.4, 1
LRD
A      #Error4_Stop:L1.3
R      #Star_Middle:L0.3, 1
EU
S      #Stop_Middle:L0.4, 1
LRD
LPS
A      #Star_Middle:L0.3
AN     #Stop_Middle:L0.4
=      #Auto_State:L0.5
LPP
A      #Star_Middle:L0.3
A      #Auto_State:L0.5
A      #E_Stop:L1.5
R      #Auto_Mode:L0.0, 6
LRD
A      Always_On:SM0.0
LPS
A      #Auto_Mode:L0.0
EU
R      #Hand_Mode:L0.1, 1
LRD
A      #Auto_Mode:L0.0
ED
R      #System_Star:L0.2, 1
LRD
A      #System_Star:L0.2
ED
R      #Auto_Mode:L0.0, 1
LRD
A      #Auto_Mode:L0.0
A      #System_Star:L0.2
R      #Hand_Mode:L0.1, 1
LPP
AN     #System_Star:L0.2
A      #Auto_Mode:L0.0
A      #Hand_Mode:L0.1
EU
R      #Auto_Mode:L0.0, 1
LRD
AN     #Hand_Mode:L0.1
AN     #Auto_Mode:L0.0
AN     #System_Error:L1.4
AN     #Stop_Middle:L0.4
AN     #Star_Middle:L0.3
AN     #Auto_State:L0.5
=      #Standby:L0.7
LRD
LD     #Error1_Stop:L1.0
O      #Error2_Stop:L1.1
O      #Error3_Stop:L1.2
O      #Error4_Stop:L1.3
ALD
EU
R      #Auto_Mode:L0.0, 4
LRD
A      #Stop_over:L1.6
EU
R      #Stop_Middle:L0.4, 1
R      #Stop_over:L1.6, 1
LPP
A      #Rest:L0.6
EU
R      #Error1_Stop:L1.0, 6
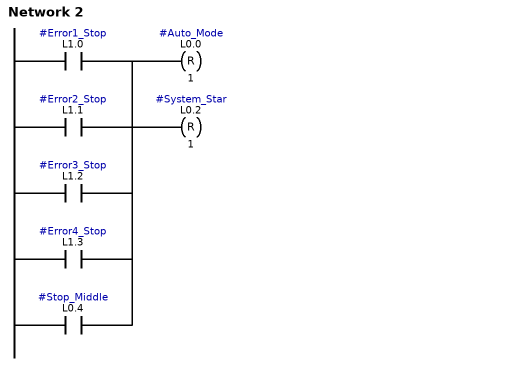
Network 2
LD     #Error1_Stop:L1.0
O      #Error2_Stop:L1.1
O      #Error3_Stop:L1.2
O      #Error4_Stop:L1.3
O      #Stop_Middle:L0.4
R      #Auto_Mode:L0.0, 1
R      #System_Star:L0.2, 1
END_SUBROUTINE_BLOCK

SUBROUTINE_BLOCK 分级机反控加料机:SBR9
TITLE=
VAR_INPUT
Sure:BOOL;	// L0.0 
Start:BOOL;	// L0.1 
InPut_A:INT;	// LW1 
Open_A:INT;	// LW3 
Close_A:INT;	// LW5 
Open_Delay:WORD;	// LW7 
Close_Delay:WORD;	// LW9 
END_VAR
VAR_IN_OUT
Motor:BOOL;	// L11.0 
END_VAR
VAR
T_Sign:BOOL;	// L11.1  超电流条件
END_VAR
BEGIN
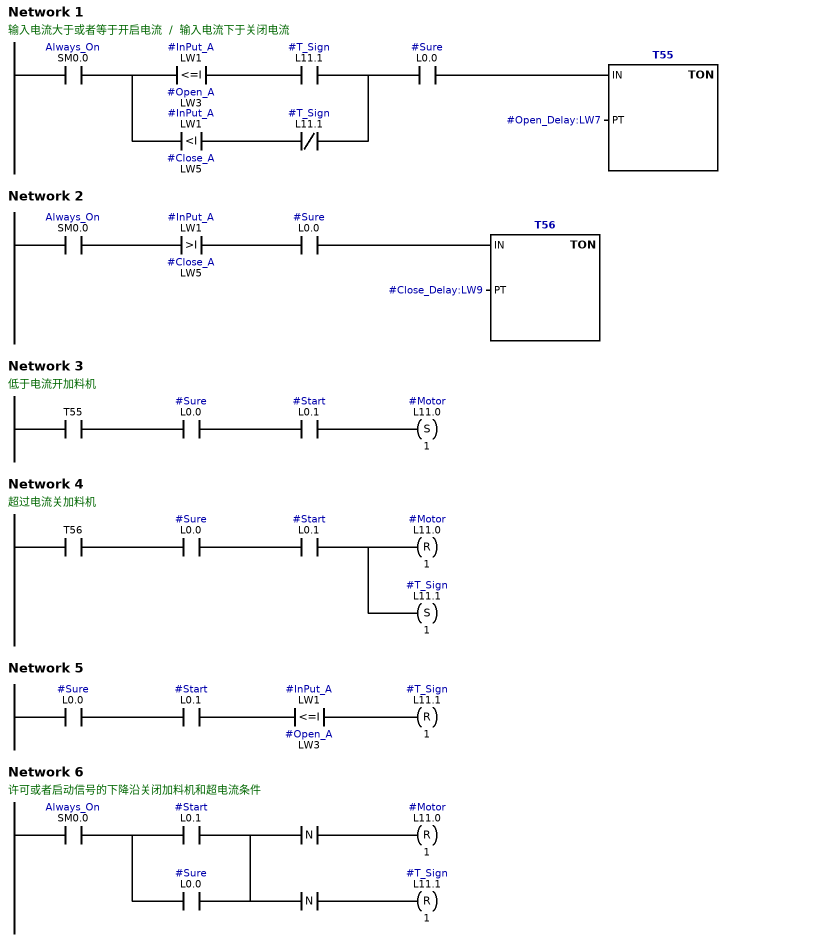
Network 1
//  输入电流大于或者等于开启电流 
//  输入电流下于关闭电流
LD     Always_On:SM0.0
LDW<=  #InPut_A:LW1, #Open_A:LW3
A      #T_Sign:L11.1
LDW<   #InPut_A:LW1, #Close_A:LW5
AN     #T_Sign:L11.1
OLD
ALD
A      #Sure:L0.0
TON    T55, #Open_Delay:LW7
Network 2
LD     Always_On:SM0.0
AW>    #InPut_A:LW1, #Close_A:LW5
A      #Sure:L0.0
TON    T56, #Close_Delay:LW9
Network 3
//  低于电流开加料机
LD     T55
A      #Sure:L0.0
A      #Start:L0.1
S      #Motor:L11.0, 1
Network 4
//  超过电流关加料机
LD     T56
A      #Sure:L0.0
A      #Start:L0.1
R      #Motor:L11.0, 1
S      #T_Sign:L11.1, 1
Network 5
LD     #Sure:L0.0
A      #Start:L0.1
AW<=   #InPut_A:LW1, #Open_A:LW3
R      #T_Sign:L11.1, 1
Network 6
//  许可或者启动信号的下降沿关闭加料机和超电流条件
LD     Always_On:SM0.0
LD     #Start:L0.1
O      #Sure:L0.0
ALD
LPS
ED
R      #Motor:L11.0, 1
LPP
ED
R      #T_Sign:L11.1, 1
END_SUBROUTINE_BLOCK

SUBROUTINE_BLOCK 手动与输出:SBR10
TITLE=
BEGIN
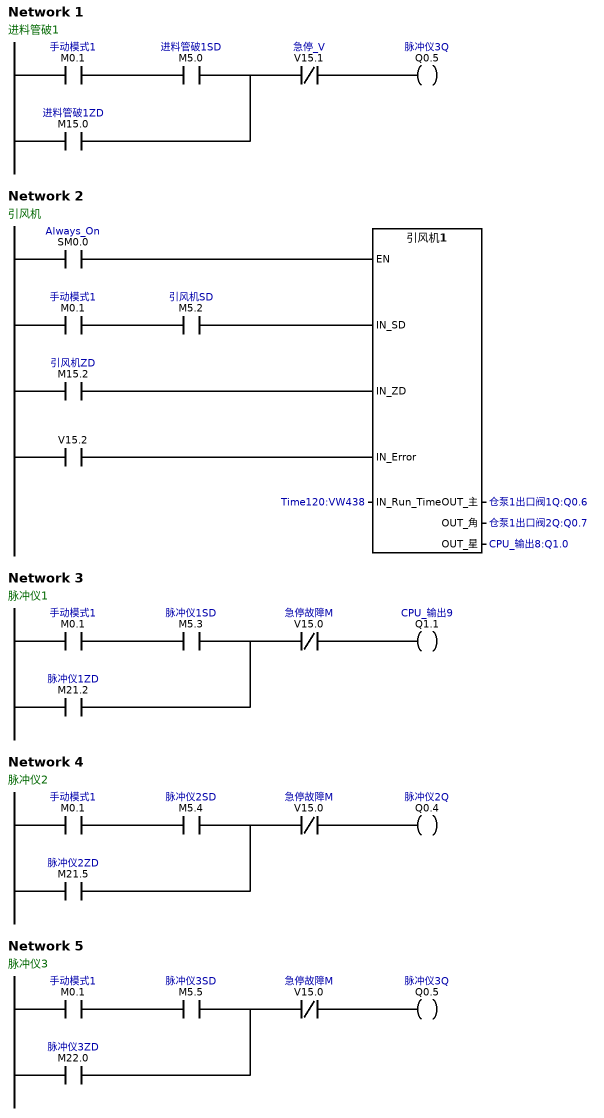
Network 1
// 进料管破1
LD     手动模式1:M0.1
A      进料管破1SD:M5.0
O      进料管破1ZD:M15.0
AN     急停_V:V15.1
=      脉冲仪3Q:Q0.5
Network 2
// 引风机
LD     Always_On:SM0.0
=      L60.0
LD     手动模式1:M0.1
A      引风机SD:M5.2
=      L63.7
LD     引风机ZD:M15.2
=      L63.6
LD     V15.2
=      L63.5
LD     L60.0
CALL   引风机1:SBR70, L63.7, L63.6, L63.5, Time120:VW438, 仓泵1出口阀1Q:Q0.6, 仓泵1出口阀2Q:Q0.7, CPU_输出8:Q1.0
Network 3
// 脉冲仪1
LD     手动模式1:M0.1
A      脉冲仪1SD:M5.3
O      脉冲仪1ZD:M21.2
AN     急停故障M:V15.0
=      CPU_输出9:Q1.1
Network 4
// 脉冲仪2
LD     手动模式1:M0.1
A      脉冲仪2SD:M5.4
O      脉冲仪2ZD:M21.5
AN     急停故障M:V15.0
=      脉冲仪2Q:Q0.4
Network 5
// 脉冲仪3
LD     手动模式1:M0.1
A      脉冲仪3SD:M5.5
O      脉冲仪3ZD:M22.0
AN     急停故障M:V15.0
=      脉冲仪3Q:Q0.5
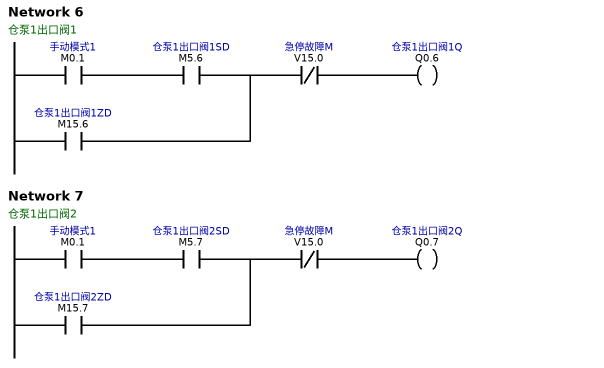
Network 6
// 仓泵1出口阀1
LD     手动模式1:M0.1
A      仓泵1出口阀1SD:M5.6
O      仓泵1出口阀1ZD:M15.6
AN     急停故障M:V15.0
=      仓泵1出口阀1Q:Q0.6
Network 7
// 仓泵1出口阀2
LD     手动模式1:M0.1
A      仓泵1出口阀2SD:M5.7
O      仓泵1出口阀2ZD:M15.7
AN     急停故障M:V15.0
=      仓泵1出口阀2Q:Q0.7
END_SUBROUTINE_BLOCK

// SBR11: protected block, not included

SUBROUTINE_BLOCK 模拟量:SBR12
TITLE=
BEGIN
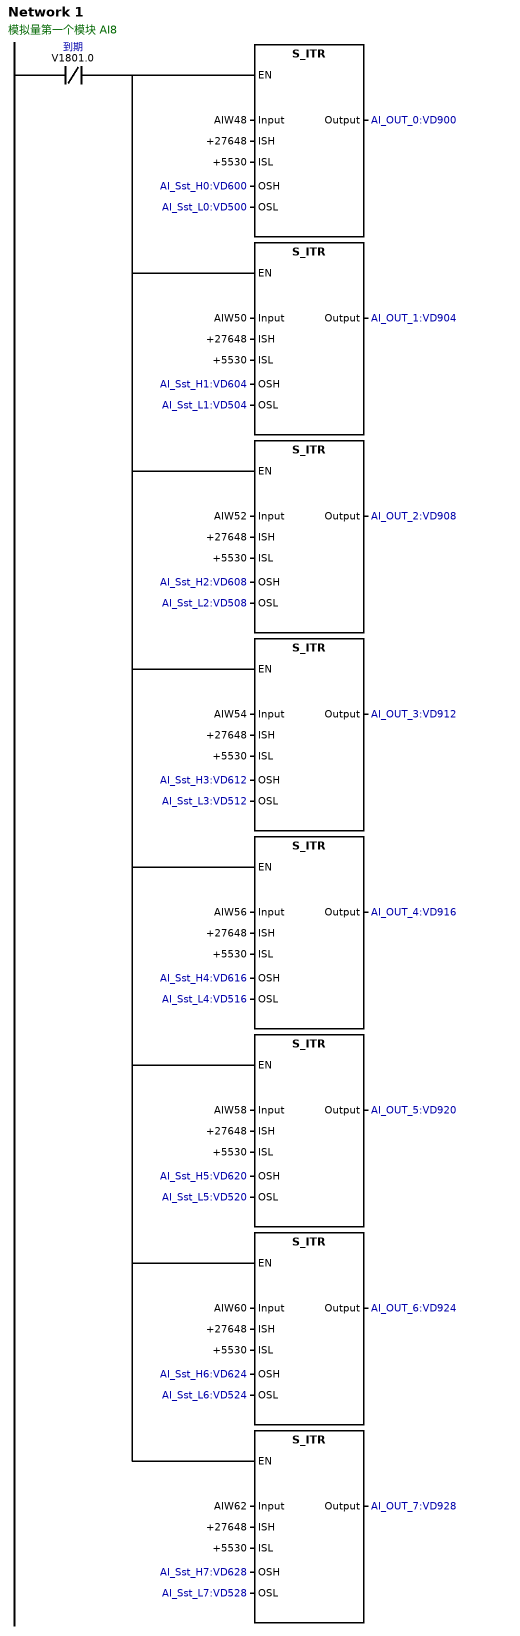
Network 1
// 模拟量第一个模块 AI8
LDN    到期:V1801.0
CALL   S_ITR:SBR6, AIW48, +27648, +5530, AI_Sst_H0:VD600, AI_Sst_L0:VD500, AI_OUT_0:VD900
CALL   S_ITR:SBR6, AIW50, +27648, +5530, AI_Sst_H1:VD604, AI_Sst_L1:VD504, AI_OUT_1:VD904
CALL   S_ITR:SBR6, AIW52, +27648, +5530, AI_Sst_H2:VD608, AI_Sst_L2:VD508, AI_OUT_2:VD908
CALL   S_ITR:SBR6, AIW54, +27648, +5530, AI_Sst_H3:VD612, AI_Sst_L3:VD512, AI_OUT_3:VD912
CALL   S_ITR:SBR6, AIW56, +27648, +5530, AI_Sst_H4:VD616, AI_Sst_L4:VD516, AI_OUT_4:VD916
CALL   S_ITR:SBR6, AIW58, +27648, +5530, AI_Sst_H5:VD620, AI_Sst_L5:VD520, AI_OUT_5:VD920
CALL   S_ITR:SBR6, AIW60, +27648, +5530, AI_Sst_H6:VD624, AI_Sst_L6:VD524, AI_OUT_6:VD924
CALL   S_ITR:SBR6, AIW62, +27648, +5530, AI_Sst_H7:VD628, AI_Sst_L7:VD528, AI_OUT_7:VD928
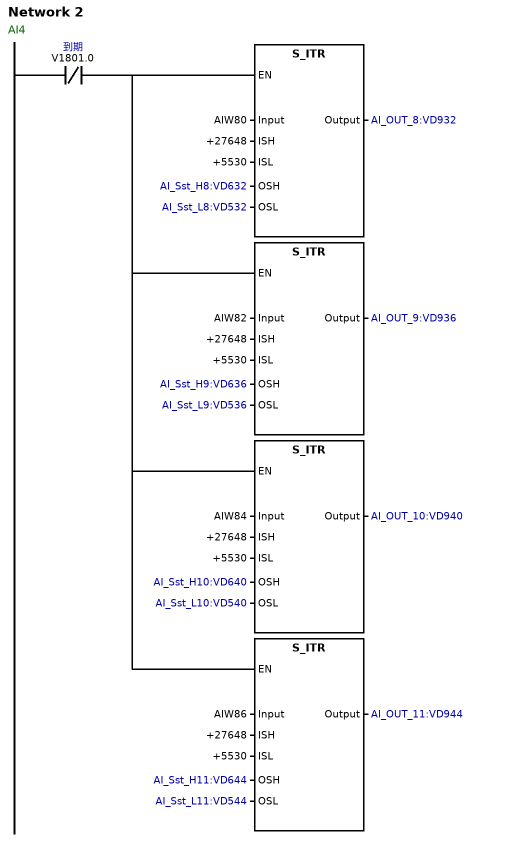
Network 2
// AI4
LDN    到期:V1801.0
CALL   S_ITR:SBR6, AIW80, +27648, +5530, AI_Sst_H8:VD632, AI_Sst_L8:VD532, AI_OUT_8:VD932
CALL   S_ITR:SBR6, AIW82, +27648, +5530, AI_Sst_H9:VD636, AI_Sst_L9:VD536, AI_OUT_9:VD936
CALL   S_ITR:SBR6, AIW84, +27648, +5530, AI_Sst_H10:VD640, AI_Sst_L10:VD540, AI_OUT_10:VD940
CALL   S_ITR:SBR6, AIW86, +27648, +5530, AI_Sst_H11:VD644, AI_Sst_L11:VD544, AI_OUT_11:VD944
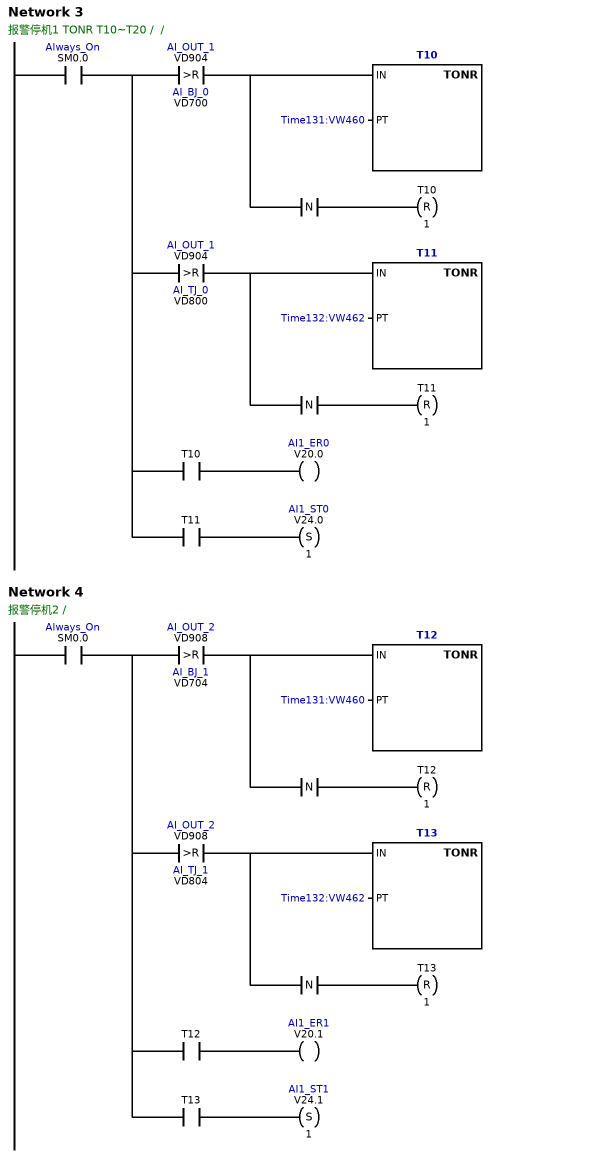
Network 3
// 报警停机1 TONR T10~T20
// 
// 
LD     Always_On:SM0.0
LPS
AR>    AI_OUT_1:VD904, AI_BJ_0:VD700
TONR   T10, Time131:VW460
ED
R      T10, 1
LRD
AR>    AI_OUT_1:VD904, AI_TJ_0:VD800
TONR   T11, Time132:VW462
ED
R      T11, 1
LPP
LPS
A      T10
=      AI1_ER0:V20.0
LPP
A      T11
S      AI1_ST0:V24.0, 1
Network 4
// 报警停机2
// 
LD     Always_On:SM0.0
LPS
AR>    AI_OUT_2:VD908, AI_BJ_1:VD704
TONR   T12, Time131:VW460
ED
R      T12, 1
LRD
AR>    AI_OUT_2:VD908, AI_TJ_1:VD804
TONR   T13, Time132:VW462
ED
R      T13, 1
LPP
LPS
A      T12
=      AI1_ER1:V20.1
LPP
A      T13
S      AI1_ST1:V24.1, 1
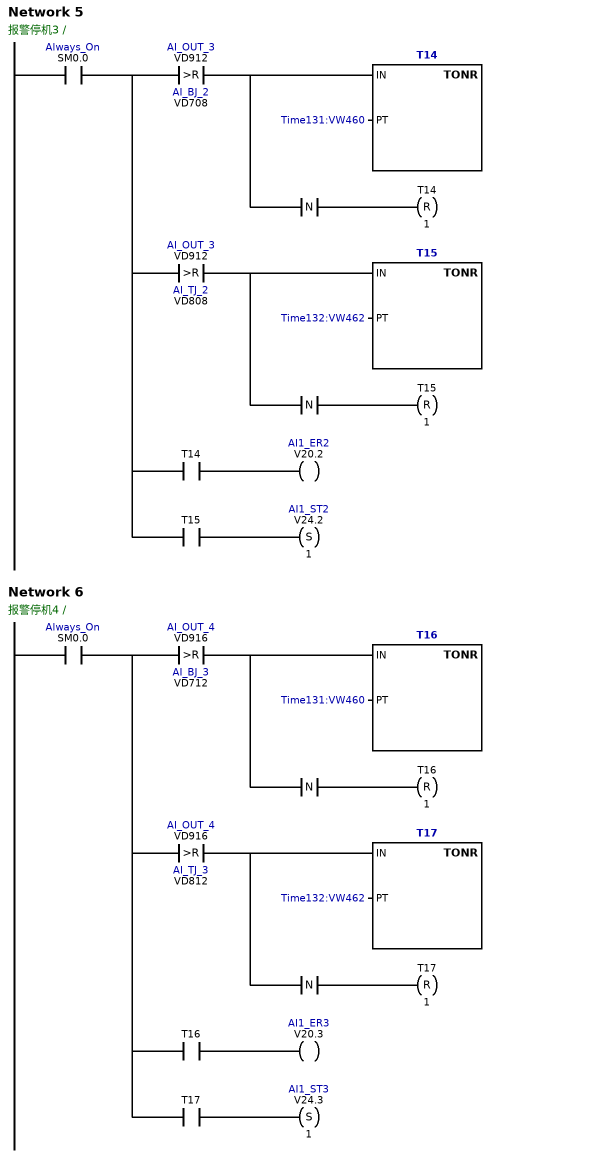
Network 5
// 报警停机3
// 
LD     Always_On:SM0.0
LPS
AR>    AI_OUT_3:VD912, AI_BJ_2:VD708
TONR   T14, Time131:VW460
ED
R      T14, 1
LRD
AR>    AI_OUT_3:VD912, AI_TJ_2:VD808
TONR   T15, Time132:VW462
ED
R      T15, 1
LPP
LPS
A      T14
=      AI1_ER2:V20.2
LPP
A      T15
S      AI1_ST2:V24.2, 1
Network 6
// 报警停机4
// 
LD     Always_On:SM0.0
LPS
AR>    AI_OUT_4:VD916, AI_BJ_3:VD712
TONR   T16, Time131:VW460
ED
R      T16, 1
LRD
AR>    AI_OUT_4:VD916, AI_TJ_3:VD812
TONR   T17, Time132:VW462
ED
R      T17, 1
LPP
LPS
A      T16
=      AI1_ER3:V20.3
LPP
A      T17
S      AI1_ST3:V24.3, 1
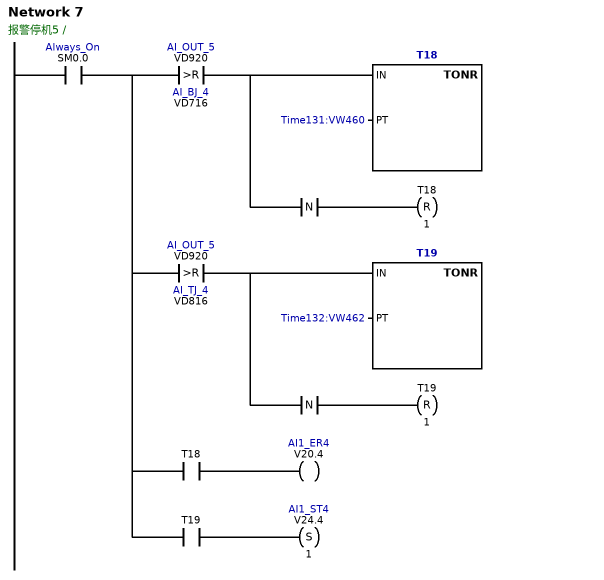
Network 7
// 报警停机5
// 
LD     Always_On:SM0.0
LPS
AR>    AI_OUT_5:VD920, AI_BJ_4:VD716
TONR   T18, Time131:VW460
ED
R      T18, 1
LRD
AR>    AI_OUT_5:VD920, AI_TJ_4:VD816
TONR   T19, Time132:VW462
ED
R      T19, 1
LPP
LPS
A      T18
=      AI1_ER4:V20.4
LPP
A      T19
S      AI1_ST4:V24.4, 1
END_SUBROUTINE_BLOCK

SUBROUTINE_BLOCK 负压控制程序:SBR13
TITLE=
VAR_INPUT
Error:BOOL;	// L0.0 
Start:BOOL;	// L0.1 
Analog_OUT:REAL;	// LD1 
Analog_L:REAL;	// LD5 
Analog_M:REAL;	// LD9 
Analog_H:REAL;	// LD13 
TIME0:WORD;	// LW17 
END_VAR
VAR_IN_OUT
Exhaust:BOOL;	// L19.0 
Fill_gas:BOOL;	// L19.1 
END_VAR
BEGIN
